C09107=1020.739,297.786,363.988,170.220,49.597,159.600
C09108=1020.733,297.538,364.020,170.215,49.601,159.600
C09109=1020.726,297.291,364.052,170.211,49.603,159.600
C09110=1020.720,297.042,364.084,170.205,49.607,159.600
C09111=1020.713,296.795,364.116,170.200,49.610,159.600
C09112=1020.707,296.547,364.149,170.195,49.613,159.600
C09113=1020.700,296.299,364.180,170.189,49.617,159.600
C09114=1020.694,296.051,364.212,170.184,49.620,159.599
C09115=1020.689,295.804,364.244,170.179,49.623,159.599
C09116=1020.682,295.556,364.276,170.174,49.627,159.599
C09117=1020.676,295.308,364.308,170.168,49.630,159.599
C09118=1020.669,295.061,364.340,170.163,49.633,159.599
C09119=1020.663,294.812,364.372,170.158,49.637,159.599
C09120=1020.657,294.564,364.404,170.153,49.640,159.599
C09121=1020.650,294.316,364.435,170.148,49.643,159.599
C09122=1020.644,294.068,364.467,170.143,49.647,159.599
C09123=1020.638,293.821,364.499,170.138,49.650,159.599
C09124=1020.632,293.592,364.529,170.133,49.653,159.599
C09125=1020.627,293.362,364.558,170.128,49.656,159.599
C09126=1020.620,293.133,364.587,170.123,49.659,159.599
C09127=1020.614,292.904,364.616,170.119,49.662,159.599
C09128=1020.608,292.674,364.645,170.113,49.666,159.599
C09129=1020.603,292.445,364.675,170.110,49.669,159.599
C09130=1020.596,292.216,364.704,170.104,49.673,159.599
C09131=1020.590,291.986,364.732,170.100,49.675,159.599
C09132=1020.584,291.738,364.764,170.095,49.679,159.599
C09133=1020.578,291.490,364.796,170.090,49.683,159.599
C09134=1020.571,291.242,364.827,170.084,49.686,159.599
C09135=1020.565,290.995,364.858,170.079,49.690,159.599
C09136=1020.558,290.747,364.890,170.074,49.693,159.599
C09137=1020.552,290.499,364.921,170.069,49.697,159.599
C09138=1020.545,290.251,364.952,170.064,49.700,159.599
C09139=1020.539,290.004,364.983,170.059,49.704,159.599
C09140=1020.533,289.756,365.015,170.054,49.707,159.599
C09141=1020.526,289.507,365.046,170.049,49.711,159.599
C09142=1020.520,289.259,365.077,170.044,49.715,159.599
C09143=1020.514,289.012,365.108,170.038,49.719,159.599
C09144=1020.507,288.763,365.139,170.034,49.722,159.599
C09145=1020.500,288.515,365.170,170.028,49.726,159.599
C09146=1020.494,288.268,365.202,170.023,49.730,159.599
C09147=1020.488,288.020,365.232,170.018,49.734,159.599
C09148=1020.481,287.772,365.264,170.014,49.736,159.599
C09149=1020.474,287.524,365.295,170.009,49.740,159.599
C09150=1020.469,287.276,365.325,170.004,49.744,159.599
C09151=1020.462,287.028,365.357,169.999,49.748,159.599
C09152=1020.455,286.780,365.388,169.994,49.752,159.599
C09153=1020.449,286.533,365.419,169.989,49.755,159.599
C09154=1020.443,286.284,365.449,169.984,49.759,159.599
C09155=1020.436,286.036,365.481,169.979,49.763,159.599
C09156=1020.430,285.788,365.511,169.974,49.767,159.599
C09157=1020.424,285.540,365.543,169.969,49.771,159.599
C09158=1020.417,285.292,365.573,169.964,49.774,159.599
C09159=1020.411,285.045,365.604,169.959,49.778,159.599
C09160=1020.405,284.796,365.635,169.954,49.782,159.600
C09161=1020.399,284.548,365.665,169.949,49.786,159.599
C09162=1020.392,284.300,365.697,169.944,49.789,159.600
C09163=1020.386,284.052,365.728,169.939,49.793,159.600
C09164=1020.379,283.804,365.757,169.934,49.797,159.600
C09165=1020.373,283.556,365.788,169.929,49.801,159.600
C09166=1020.367,283.309,365.819,169.924,49.805,159.600
C09167=1020.360,283.060,365.850,169.919,49.809,159.600
C09168=1020.354,282.812,365.881,169.914,49.813,159.600
C09169=1020.347,282.564,365.910,169.909,49.817,159.600
C09170=1020.341,282.316,365.942,169.904,49.821,159.600
C09171=1020.335,282.068,365.972,169.899,49.825,159.600
C09172=1020.328,281.820,366.003,169.895,49.829,159.600
C09173=1020.322,281.572,366.033,169.890,49.833,159.600
C09174=1020.315,281.324,366.063,169.886,49.836,159.601
C09175=1020.309,281.076,366.094,169.881,49.840,159.601
C09176=1020.303,280.827,366.124,169.876,49.845,159.601
C09177=1020.297,280.580,366.155,169.871,49.849,159.601
C09178=1020.290,280.332,366.186,169.866,49.853,159.601
C09179=1020.284,280.084,366.216,169.861,49.857,159.601
C09180=1020.278,279.836,366.247,169.856,49.861,159.601
C09181=1020.272,279.588,366.277,169.852,49.865,159.601
C09182=1020.265,279.340,366.307,169.847,49.868,159.602
C09183=1020.259,279.092,366.337,169.842,49.872,159.602
C09184=1020.254,278.869,366.365,169.838,49.876,159.602
C09185=1020.247,278.645,366.392,169.833,49.880,159.602
C09186=1020.242,278.422,366.419,169.829,49.884,159.602
C09187=1020.237,278.199,366.447,169.825,49.887,159.602
C09188=1020.231,277.976,366.474,169.820,49.891,159.602
C09189=1020.226,277.753,366.501,169.816,49.895,159.603
C09190=1020.219,277.529,366.528,169.812,49.898,159.603
C09191=1020.214,277.306,366.556,169.807,49.902,159.603
C09192=1020.209,277.058,366.586,169.802,49.906,159.603
C09193=1020.201,276.810,366.616,169.797,49.910,159.603
C09194=1020.196,276.562,366.647,169.792,49.914,159.603
C09195=1020.189,276.314,366.676,169.788,49.919,159.603
C09196=1020.183,276.066,366.707,169.783,49.923,159.603
C09197=1020.176,275.818,366.736,169.778,49.927,159.604
C09198=1020.171,275.570,366.766,169.774,49.931,159.604
C09199=1020.163,275.322,366.797,169.769,49.935,159.604
C09200=1020.158,275.073,366.826,169.764,49.940,159.604
C09201=1020.152,274.825,366.857,169.759,49.944,159.604
C09202=1020.145,274.577,366.887,169.755,49.948,159.604
C09203=1020.139,274.329,366.916,169.751,49.952,159.605
C09204=1020.133,274.081,366.946,169.746,49.957,159.605
C09205=1020.126,273.833,366.977,169.741,49.961,159.605
C09206=1020.120,273.584,367.006,169.737,49.965,159.605
C09207=1020.114,273.337,367.036,169.732,49.969,159.605
C09208=1020.107,273.088,367.066,169.727,49.974,159.606
C09209=1020.102,272.840,367.096,169.722,49.978,159.606
C09210=1020.095,272.592,367.126,169.718,49.982,159.606
C09211=1020.090,272.344,367.155,169.713,49.986,159.606
C09212=1020.082,272.096,367.185,169.708,49.991,159.606
C09213=1020.076,271.848,367.214,169.704,49.995,159.607
C09214=1020.070,271.600,367.245,169.699,49.999,159.607
C09215=1020.064,271.352,367.274,169.694,50.004,159.607
C09216=1020.058,271.103,367.304,169.690,50.009,159.607
C09217=1020.051,270.855,367.334,169.685,50.013,159.607
C09218=1020.046,270.607,367.363,169.680,50.017,159.608
C09219=1020.039,270.359,367.393,169.676,50.022,159.608
C09220=1020.033,270.111,367.422,169.671,50.026,159.608
C09221=1020.027,269.862,367.453,169.666,50.030,159.608
C09222=1020.020,269.614,367.482,169.662,50.035,159.609
C09223=1020.015,269.366,367.511,169.657,50.039,159.609
C09224=1020.009,269.118,367.540,169.652,50.044,159.609
C09225=1020.002,268.870,367.570,169.648,50.048,159.609
C09226=1019.996,268.622,367.599,169.643,50.053,159.610
C09227=1019.990,268.373,367.629,169.638,50.057,159.610
C09228=1019.984,268.125,367.658,169.634,50.061,159.610
C09229=1019.977,267.877,367.688,169.629,50.066,159.610
C09230=1019.971,267.629,367.718,169.624,50.071,159.610
C09231=1019.965,267.381,367.747,169.620,50.075,159.611
C09232=1019.959,267.133,367.776,169.615,50.080,159.611
C09233=1019.953,266.885,367.805,169.611,50.085,159.611
C09234=1019.946,266.636,367.836,169.606,50.089,159.612
C09235=1019.940,266.388,367.865,169.602,50.094,159.612
C09236=1019.934,266.140,367.894,169.597,50.098,159.612
C09237=1019.928,265.892,367.923,169.593,50.103,159.612
C09238=1019.921,265.643,367.952,169.588,50.107,159.612
C09239=1019.916,265.395,367.981,169.583,50.112,159.613
C09240=1019.910,265.147,368.010,169.579,50.116,159.613
C09241=1019.903,264.899,368.039,169.574,50.121,159.613
C09242=1019.897,264.651,368.068,169.570,50.126,159.614
C09243=1019.891,264.402,368.097,169.565,50.131,159.614
C09244=1019.885,264.182,368.124,169.560,50.135,159.614
C09245=1019.880,263.961,368.149,169.557,50.139,159.615
C09246=1019.874,263.740,368.175,169.553,50.143,159.615
C09247=1019.868,263.519,368.201,169.548,50.147,159.615
C09248=1019.863,263.298,368.227,169.545,50.152,159.615
C09249=1019.857,263.078,368.253,169.541,50.155,159.615
C09250=1019.852,262.856,368.278,169.537,50.160,159.616
C09251=1019.846,262.636,368.304,169.533,50.164,159.616
C09252=1019.841,262.387,368.334,169.528,50.169,159.616
C09253=1019.835,262.139,368.363,169.524,50.174,159.617
C09254=1019.829,261.890,368.391,169.519,50.178,159.617
C09255=1019.822,261.642,368.420,169.515,50.183,159.617
C09256=1019.816,261.394,368.449,169.511,50.188,159.618
C09257=1019.810,261.146,368.478,169.506,50.193,159.618
C09258=1019.804,260.898,368.507,169.502,50.198,159.618
C09259=1019.798,260.649,368.536,169.497,50.202,159.619
C09260=1019.791,260.401,368.565,169.493,50.207,159.619
C09261=1019.785,260.153,368.594,169.488,50.212,159.619
C09262=1019.779,259.905,368.623,169.484,50.217,159.620
C09263=1019.773,259.656,368.651,169.478,50.222,159.620
C09264=1019.766,259.408,368.680,169.474,50.227,159.620
C09265=1019.760,259.159,368.708,169.470,50.232,159.620
C09266=1019.754,258.912,368.737,169.465,50.237,159.621
C09267=1019.748,258.664,368.764,169.461,50.242,159.621
C09268=1019.741,258.415,368.793,169.457,50.247,159.622
C09269=1019.736,258.167,368.822,169.452,50.252,159.622
C09270=1019.729,257.919,368.850,169.448,50.257,159.622
C09271=1019.723,257.670,368.879,169.444,50.262,159.623
C09272=1019.716,257.422,368.908,169.438,50.267,159.623
C09273=1019.710,257.173,368.935,169.434,50.272,159.623
C09274=1019.703,256.925,368.964,169.430,50.277,159.624
C09275=1019.697,256.677,368.993,169.425,50.282,159.624
C09276=1019.690,256.429,369.021,169.421,50.287,159.625
C09277=1019.685,256.180,369.049,169.417,50.293,159.625
C09278=1019.679,255.932,369.077,169.412,50.297,159.625
C09279=1019.672,255.684,369.106,169.408,50.303,159.626
C09280=1019.666,255.435,369.134,169.403,50.308,159.626
C09281=1019.660,255.187,369.162,169.399,50.313,159.627
C09282=1019.653,254.939,369.191,169.394,50.318,159.627
C09283=1019.647,254.690,369.219,169.390,50.323,159.627
C09284=1019.642,254.442,369.247,169.386,50.328,159.628
C09285=1019.635,254.194,369.276,169.381,50.333,159.628
C09286=1019.629,253.945,369.304,169.377,50.338,159.628
C09287=1019.623,253.697,369.332,169.373,50.343,159.629
C09288=1019.616,253.448,369.360,169.368,50.348,159.629
C09289=1019.611,253.201,369.389,169.363,50.354,159.630
C09290=1019.605,252.952,369.417,169.359,50.359,159.630
C09291=1019.598,252.704,369.445,169.355,50.364,159.631
C09292=1019.592,252.455,369.473,169.350,50.369,159.631
C09293=1019.586,252.207,369.502,169.346,50.374,159.631
C09294=1019.580,251.959,369.530,169.342,50.380,159.632
C09295=1019.574,251.710,369.558,169.338,50.385,159.632
C09296=1019.568,251.461,369.586,169.333,50.390,159.633
C09297=1019.562,251.214,369.614,169.329,50.395,159.633
C09298=1019.556,250.966,369.643,169.324,50.401,159.633
C09299=1019.550,250.717,369.671,169.320,50.406,159.634
C09300=1019.543,250.468,369.699,169.316,50.411,159.634
C09301=1019.538,250.220,369.727,169.311,50.416,159.635
C09302=1019.532,249.972,369.755,169.307,50.422,159.635
C09303=1019.525,249.723,369.783,169.303,50.427,159.636
C09304=1019.520,249.502,369.808,169.299,50.432,159.636
C09305=1019.515,249.280,369.833,169.295,50.437,159.636
C09306=1019.510,249.058,369.857,169.292,50.441,159.637
C09307=1019.504,248.837,369.883,169.287,50.446,159.637
C09308=1019.499,248.614,369.908,169.284,50.451,159.638
C09309=1019.493,248.393,369.933,169.280,50.455,159.638
C09310=1019.488,248.171,369.958,169.276,50.460,159.638
C09311=1019.483,247.950,369.983,169.272,50.465,159.639
C09312=1019.476,247.702,370.011,169.268,50.470,159.639
C09313=1019.471,247.454,370.039,169.264,50.476,159.640
C09314=1019.464,247.205,370.067,169.260,50.481,159.640
C09315=1019.458,246.956,370.094,169.256,50.486,159.641
C09316=1019.453,246.708,370.122,169.251,50.491,159.641
C09317=1019.446,246.459,370.150,169.247,50.496,159.641
C09318=1019.441,246.211,370.178,169.242,50.502,159.642
C09319=1019.435,245.962,370.206,169.238,50.508,159.642
C09320=1019.429,245.714,370.234,169.234,50.513,159.643
C09321=1019.423,245.466,370.262,169.229,50.518,159.643
C09322=1019.417,245.217,370.290,169.225,50.524,159.643
C09323=1019.411,244.969,370.318,169.221,50.529,159.644
C09324=1019.405,244.721,370.346,169.217,50.534,159.644
C09325=1019.399,244.473,370.373,169.213,50.540,159.645
C09326=1019.393,244.224,370.401,169.209,50.546,159.646
C09327=1019.388,243.976,370.429,169.204,50.551,159.646
C09328=1019.381,243.727,370.457,169.200,50.557,159.646
C09329=1019.376,243.479,370.485,169.196,50.562,159.647
C09330=1019.370,243.230,370.513,169.192,50.567,159.647
C09331=1019.364,242.982,370.540,169.188,50.573,159.648
C09332=1019.358,242.733,370.567,169.184,50.578,159.648
C09333=1019.352,242.485,370.595,169.180,50.584,159.649
C09334=1019.346,242.236,370.622,169.175,50.590,159.649
C09335=1019.340,241.989,370.650,169.171,50.595,159.650
C09336=1019.334,241.740,370.678,169.166,50.601,159.650
C09337=1019.328,241.492,370.705,169.163,50.607,159.651
C09338=1019.322,241.243,370.732,169.159,50.612,159.651
C09339=1019.316,240.994,370.760,169.153,50.618,159.652
C09340=1019.310,240.746,370.787,169.150,50.624,159.652
C09341=1019.304,240.498,370.815,169.146,50.629,159.653
C09342=1019.298,240.249,370.842,169.141,50.635,159.653
C09343=1019.292,240.001,370.870,169.138,50.641,159.654
C09344=1019.286,239.753,370.896,169.133,50.646,159.654
C09345=1019.280,239.504,370.925,169.129,50.652,159.655
C09346=1019.275,239.256,370.951,169.125,50.658,159.656
C09347=1019.268,239.007,370.979,169.121,50.663,159.656
C09348=1019.262,238.759,371.006,169.117,50.669,159.657
C09349=1019.256,238.510,371.034,169.112,50.675,159.657
C09350=1019.250,238.262,371.061,169.108,50.681,159.658
C09351=1019.245,238.013,371.087,169.104,50.686,159.658
C09352=1019.238,237.765,371.115,169.100,50.692,159.659
C09353=1019.232,237.517,371.142,169.095,50.698,159.659
C09354=1019.226,237.268,371.169,169.091,50.704,159.660
C09355=1019.220,237.020,371.196,169.087,50.710,159.660
C09356=1019.214,236.771,371.223,169.083,50.716,159.661
C09357=1019.208,236.522,371.250,169.079,50.722,159.662
C09358=1019.202,236.274,371.276,169.075,50.727,159.662
C09359=1019.195,236.026,371.304,169.071,50.734,159.663
C09360=1019.189,235.777,371.331,169.066,50.739,159.663
C09361=1019.184,235.529,371.357,169.062,50.745,159.664
C09362=1019.177,235.280,371.384,169.059,50.751,159.664
C09363=1019.171,235.032,371.412,169.054,50.757,159.665
C09364=1019.166,234.807,371.436,169.051,50.763,159.666
C09365=1019.160,234.581,371.460,169.047,50.768,159.666
C09366=1019.155,234.356,371.485,169.043,50.774,159.667
C09367=1019.150,234.132,371.509,169.039,50.779,159.667
C09368=1019.145,233.907,371.533,169.035,50.784,159.668
C09369=1019.139,233.682,371.558,169.031,50.790,159.668
C09370=1019.134,233.457,371.582,169.029,50.795,159.669
C09371=1019.128,233.232,371.606,169.024,50.801,159.669
C09372=1019.122,232.983,371.633,169.021,50.807,159.670
C09373=1019.116,232.735,371.660,169.016,50.812,159.670
C09374=1019.110,232.487,371.686,169.012,50.819,159.671
C09375=1019.104,232.238,371.713,169.008,50.825,159.672
C09376=1019.098,231.989,371.740,169.004,50.831,159.672
C09377=1019.092,231.741,371.767,169.000,50.837,159.673
C09378=1019.086,231.493,371.794,168.996,50.843,159.673
C09379=1019.080,231.245,371.821,168.992,50.849,159.674
C09380=1019.074,230.996,371.848,168.987,50.855,159.675
C09381=1019.068,230.747,371.874,168.984,50.861,159.675
C09382=1019.062,230.499,371.901,168.980,50.867,159.676
C09383=1019.057,230.251,371.928,168.975,50.874,159.676
C09384=1019.050,230.001,371.955,168.972,50.880,159.677
C09385=1019.044,229.753,371.981,168.968,50.886,159.678
C09386=1019.039,229.504,372.007,168.963,50.892,159.678
C09387=1019.033,229.256,372.034,168.959,50.898,159.679
C09388=1019.027,229.007,372.061,168.955,50.904,159.680
C09389=1019.020,228.759,372.087,168.951,50.910,159.680
C09390=1019.015,228.510,372.114,168.947,50.916,159.681
C09391=1019.009,228.262,372.140,168.943,50.922,159.681
C09392=1019.003,228.014,372.167,168.939,50.929,159.682
C09393=1018.997,227.765,372.194,168.935,50.935,159.683
C09394=1018.992,227.516,372.220,168.932,50.942,159.684
C09395=1018.985,227.268,372.246,168.927,50.948,159.684
C09396=1018.979,227.019,372.273,168.923,50.954,159.685
C09397=1018.973,226.771,372.299,168.919,50.961,159.685
C09398=1018.968,226.522,372.325,168.915,50.967,159.686
C09399=1018.961,226.274,372.351,168.911,50.973,159.687
C09400=1018.955,226.025,372.378,168.906,50.979,159.687
C09401=1018.950,225.777,372.405,168.903,50.985,159.688
C09402=1018.943,225.528,372.430,168.899,50.993,159.689
C09403=1018.937,225.279,372.457,168.895,50.999,159.689
C09404=1018.931,225.031,372.482,168.890,51.005,159.690
C09405=1018.925,224.782,372.509,168.886,51.011,159.691
C09406=1018.919,224.534,372.536,168.883,51.018,159.692
C09407=1018.913,224.285,372.561,168.879,51.024,159.692
C09408=1018.907,224.037,372.588,168.875,51.031,159.693
C09409=1018.901,223.788,372.613,168.871,51.038,159.694
C09410=1018.895,223.539,372.640,168.867,51.044,159.694
C09411=1018.889,223.290,372.666,168.862,51.050,159.695
C09412=1018.883,223.042,372.692,168.859,51.056,159.695
C09413=1018.877,222.793,372.718,168.855,51.063,159.696
C09414=1018.871,222.545,372.744,168.851,51.070,159.697
C09415=1018.865,222.296,372.770,168.847,51.076,159.698
C09416=1018.859,222.048,372.796,168.843,51.083,159.698
C09417=1018.853,221.799,372.822,168.839,51.089,159.699
C09418=1018.847,221.551,372.848,168.835,51.096,159.700
C09419=1018.841,221.302,372.874,168.831,51.102,159.700
C09420=1018.835,221.054,372.900,168.826,51.109,159.701
C09421=1018.830,220.805,372.926,168.823,51.116,159.702
C09422=1018.824,220.557,372.952,168.818,51.122,159.702
C09423=1018.818,220.308,372.978,168.815,51.129,159.703
C09424=1018.812,220.079,373.002,168.811,51.135,159.704
C09425=1018.807,219.850,373.026,168.808,51.141,159.705
C09426=1018.801,219.621,373.050,168.804,51.147,159.705
C09427=1018.796,219.392,373.074,168.801,51.153,159.706
C09428=1018.790,219.163,373.098,168.796,51.159,159.706
C09429=1018.785,218.933,373.122,168.793,51.165,159.707
C09430=1018.779,218.704,373.146,168.789,51.171,159.708
C09431=1018.774,218.475,373.170,168.785,51.177,159.708
C09432=1018.768,218.226,373.196,168.782,51.184,159.709
C09433=1018.762,217.978,373.221,168.778,51.191,159.710
C09434=1018.757,217.730,373.246,168.774,51.197,159.711
C09435=1018.750,217.482,373.272,168.770,51.204,159.712
C09436=1018.745,217.233,373.298,168.767,51.211,159.712
C09437=1018.738,216.984,373.324,168.762,51.218,159.713
C09438=1018.732,216.735,373.349,168.758,51.225,159.714
C09439=1018.727,216.486,373.375,168.755,51.232,159.715
C09440=1018.720,216.238,373.401,168.750,51.238,159.715
C09441=1018.714,215.990,373.426,168.747,51.245,159.716
C09442=1018.708,215.741,373.452,168.742,51.252,159.717
C09443=1018.702,215.492,373.478,168.739,51.259,159.718
C09444=1018.696,215.243,373.503,168.735,51.265,159.718
C09445=1018.690,214.995,373.528,168.730,51.273,159.719
C09446=1018.684,214.746,373.554,168.727,51.279,159.720
C09447=1018.678,214.497,373.580,168.723,51.287,159.721
C09448=1018.673,214.249,373.605,168.720,51.293,159.722
C09449=1018.666,214.000,373.630,168.715,51.300,159.722
C09450=1018.661,213.752,373.657,168.712,51.307,159.723
C09451=1018.654,213.503,373.682,168.707,51.314,159.724
C09452=1018.648,213.255,373.707,168.703,51.321,159.725
C09453=1018.643,213.006,373.733,168.700,51.328,159.725
C09454=1018.637,212.757,373.759,168.696,51.335,159.726
C09455=1018.630,212.508,373.784,168.692,51.341,159.727
C09456=1018.625,212.260,373.809,168.688,51.349,159.728
C09457=1018.619,212.011,373.835,168.684,51.356,159.728
C09458=1018.613,211.763,373.860,168.680,51.363,159.729
C09459=1018.607,211.514,373.885,168.676,51.370,159.730
C09460=1018.601,211.265,373.911,168.673,51.377,159.731
C09461=1018.596,211.017,373.936,168.669,51.384,159.732
C09462=1018.590,210.768,373.962,168.664,51.391,159.733
C09463=1018.584,210.519,373.986,168.661,51.398,159.733
C09464=1018.578,210.270,374.012,168.657,51.405,159.734
C09465=1018.572,210.021,374.038,168.654,51.412,159.735
C09466=1018.566,209.774,374.063,168.650,51.419,159.736
C09467=1018.560,209.525,374.088,168.645,51.426,159.737
C09468=1018.554,209.276,374.113,168.642,51.433,159.738
C09469=1018.548,209.028,374.139,168.638,51.440,159.738
C09470=1018.542,208.778,374.163,168.634,51.448,159.739
C09471=1018.537,208.530,374.189,168.631,51.454,159.740
C09472=1018.531,208.281,374.214,168.626,51.462,159.741
C09473=1018.525,208.033,374.239,168.622,51.469,159.741
C09474=1018.518,207.784,374.265,168.618,51.477,159.742
C09475=1018.513,207.535,374.289,168.615,51.484,159.743
C09476=1018.507,207.287,374.314,168.611,51.491,159.744
C09477=1018.501,207.038,374.340,168.607,51.498,159.745
C09478=1018.495,206.789,374.364,168.603,51.505,159.746
C09479=1018.489,206.541,374.389,168.600,51.513,159.747
C09480=1018.483,206.292,374.415,168.595,51.520,159.748
C09481=1018.477,206.043,374.439,168.591,51.527,159.748
C09482=1018.472,205.795,374.464,168.588,51.534,159.749
C09483=1018.465,205.546,374.490,168.584,51.542,159.750
C09484=1018.460,205.317,374.512,168.581,51.548,159.751
C09485=1018.454,205.087,374.535,168.577,51.555,159.752
C09486=1018.449,204.858,374.559,168.573,51.562,159.752
C09487=1018.444,204.629,374.581,168.570,51.569,159.753
C09488=1018.438,204.400,374.603,168.566,51.575,159.754
C09489=1018.432,204.171,374.626,168.563,51.582,159.755
C09490=1018.426,203.942,374.650,168.559,51.589,159.756
C09491=1018.400,202.697,374.768,168.087,51.498,159.649
C09492=1018.396,202.448,374.791,168.082,51.506,159.650
C09493=1018.390,202.199,374.814,168.078,51.514,159.651
C09494=1018.385,201.950,374.837,168.073,51.523,159.652
C09495=1018.381,201.701,374.860,168.069,51.532,159.653
C09496=1018.376,201.452,374.883,168.064,51.540,159.653
C09497=1018.371,201.204,374.906,168.060,51.548,159.654
C09498=1018.366,200.954,374.929,168.055,51.556,159.655
C09499=1018.361,200.705,374.953,168.051,51.565,159.656
C09500=1018.356,200.457,374.976,168.046,51.573,159.657
C09501=1018.351,200.208,374.999,168.041,51.582,159.658
C09502=1018.346,199.959,375.022,168.037,51.590,159.659
C09503=1018.341,199.710,375.045,168.033,51.599,159.660
C09504=1018.336,199.461,375.069,168.028,51.607,159.661
C09505=1018.332,199.212,375.091,168.023,51.616,159.662
C09506=1018.326,198.963,375.114,168.019,51.624,159.663
C09507=1018.321,198.715,375.137,168.014,51.632,159.663
C09508=1018.316,198.465,375.160,168.010,51.641,159.664
C09509=1018.311,198.217,375.182,168.005,51.649,159.665
C09510=1018.305,197.968,375.205,168.001,51.658,159.666
C09511=1018.301,197.718,375.228,167.997,51.666,159.667
C09512=1018.295,197.470,375.250,167.992,51.675,159.668
C09513=1018.290,197.221,375.273,167.988,51.684,159.669
C09514=1018.286,196.972,375.296,167.983,51.693,159.670
C09515=1018.280,196.723,375.319,167.978,51.701,159.671
C09516=1018.275,196.474,375.341,167.975,51.710,159.672
C09517=1018.270,196.225,375.364,167.970,51.718,159.673
C09518=1018.265,195.976,375.386,167.966,51.727,159.674
C09519=1018.259,195.727,375.409,167.961,51.735,159.675
C09520=1018.254,195.479,375.432,167.956,51.744,159.676
C09521=1018.250,195.229,375.454,167.953,51.752,159.677
C09522=1018.245,194.981,375.477,167.948,51.761,159.678
C09523=1018.239,194.732,375.499,167.943,51.770,159.678
C09524=1018.235,194.483,375.522,167.939,51.779,159.679
C09525=1018.229,194.234,375.545,167.935,51.787,159.680
C09526=1018.224,193.985,375.567,167.931,51.796,159.681
C09527=1018.219,193.736,375.590,167.926,51.804,159.682
C09528=1018.215,193.487,375.612,167.922,51.813,159.683
C09529=1018.210,193.239,375.635,167.918,51.821,159.684
C09530=1018.205,192.989,375.657,167.913,51.830,159.685
C09531=1018.200,192.741,375.680,167.908,51.838,159.686
C09532=1018.194,192.491,375.702,167.905,51.847,159.687
C09533=1018.189,192.243,375.725,167.900,51.856,159.688
C09534=1018.185,191.994,375.747,167.896,51.865,159.689
C09535=1018.180,191.744,375.769,167.892,51.873,159.690
C09536=1018.175,191.496,375.792,167.887,51.882,159.691
C09537=1018.170,191.246,375.815,167.883,51.890,159.692
C09538=1018.165,190.998,375.837,167.879,51.899,159.693
C09539=1018.160,190.749,375.859,167.874,51.907,159.694
C09540=1018.155,190.499,375.882,167.870,51.916,159.695
C09541=1018.150,190.251,375.905,167.866,51.924,159.696
C09542=1018.145,190.002,375.927,167.862,51.933,159.697
C09543=1018.140,189.753,375.949,167.857,51.941,159.698
C09544=1018.136,189.504,375.971,167.854,51.950,159.699
C09545=1018.131,189.256,375.994,167.849,51.959,159.699
C09546=1018.125,189.006,376.016,167.845,51.968,159.701
C09547=1018.121,188.757,376.038,167.841,51.976,159.702
C09548=1018.116,188.509,376.061,167.836,51.985,159.702
C09549=1018.111,188.259,376.083,167.832,51.994,159.704
C09550=1018.106,188.010,376.106,167.828,52.002,159.704
C09551=1018.102,187.761,376.128,167.824,52.011,159.705
C09552=1018.096,187.481,376.153,167.819,52.020,159.706
C09553=1018.090,187.199,376.178,167.814,52.030,159.708
C09554=1018.085,186.919,376.203,167.810,52.039,159.709
C09555=1018.080,186.638,376.228,167.805,52.049,159.710
C09556=1018.075,186.390,376.251,167.801,52.058,159.711
C09557=1018.070,186.140,376.273,167.797,52.066,159.712
C09558=1018.065,185.892,376.295,167.793,52.075,159.713
C09559=1018.060,185.643,376.317,167.789,52.083,159.714
C09560=1018.055,185.394,376.339,167.785,52.093,159.715
C09561=1018.051,185.145,376.361,167.781,52.101,159.716
C09562=1018.046,184.896,376.384,167.776,52.110,159.717
C09563=1018.041,184.647,376.406,167.772,52.118,159.717
C09564=1018.037,184.398,376.429,167.768,52.127,159.719
C09565=1018.032,184.149,376.451,167.764,52.135,159.719
C09566=1018.027,183.900,376.472,167.760,52.144,159.721
C09567=1018.022,183.651,376.495,167.755,52.152,159.721
C09568=1018.018,183.402,376.517,167.752,52.161,159.723
C09569=1018.013,183.153,376.539,167.747,52.170,159.723
C09570=1018.008,182.904,376.561,167.744,52.178,159.724
C09571=1018.003,182.655,376.583,167.739,52.187,159.725
C09572=1017.999,182.406,376.605,167.736,52.195,159.726
C09573=1017.994,182.157,376.627,167.731,52.204,159.727
C09574=1017.989,181.908,376.649,167.728,52.213,159.728
C09575=1017.984,181.659,376.671,167.723,52.222,159.729
C09576=1017.979,181.410,376.693,167.719,52.231,159.730
C09577=1017.974,181.161,376.714,167.715,52.239,159.731
C09578=1017.968,180.912,376.736,167.711,52.248,159.732
C09579=1017.964,180.663,376.758,167.707,52.257,159.733
C09580=1017.958,180.414,376.778,167.703,52.266,159.735
C09581=1017.954,180.165,376.800,167.699,52.275,159.736
C09582=1017.949,179.916,376.822,167.695,52.284,159.737
C09583=1017.943,179.667,376.842,167.692,52.293,159.738
C09584=1017.938,179.417,376.865,167.687,52.301,159.739
C09585=1017.934,179.168,376.886,167.682,52.310,159.740
C09586=1017.928,178.919,376.907,167.679,52.319,159.741
C09587=1017.923,178.671,376.929,167.675,52.328,159.742
C09588=1017.918,178.422,376.949,167.672,52.337,159.743
C09589=1017.913,178.173,376.971,167.667,52.346,159.744
C09590=1017.909,177.923,376.993,167.663,52.355,159.745
C09591=1017.903,177.675,377.014,167.659,52.364,159.746
C09592=1017.898,177.426,377.036,167.655,52.373,159.747
C09593=1017.893,177.176,377.057,167.651,52.382,159.748
C09594=1017.887,176.927,377.078,167.647,52.391,159.749
C09595=1017.883,176.678,377.100,167.643,52.400,159.750
C09596=1017.878,176.429,377.121,167.640,52.409,159.751
C09597=1017.873,176.180,377.142,167.635,52.418,159.752
C09598=1017.868,175.931,377.164,167.631,52.426,159.753
C09599=1017.863,175.682,377.184,167.627,52.435,159.754
C09600=1017.858,175.433,377.206,167.623,52.444,159.755
C09601=1017.853,175.184,377.227,167.620,52.453,159.756
C09602=1017.848,174.935,377.249,167.616,52.462,159.757
C09603=1017.843,174.686,377.270,167.612,52.471,159.759
C09604=1017.839,174.437,377.292,167.608,52.480,159.760
C09605=1017.833,174.188,377.312,167.603,52.488,159.760
C09606=1017.828,173.939,377.334,167.600,52.497,159.762
C09607=1017.823,173.690,377.355,167.596,52.506,159.763
C09608=1017.819,173.440,377.376,167.593,52.515,159.764
C09609=1017.814,173.192,377.398,167.588,52.524,159.765
C09610=1017.809,172.943,377.418,167.585,52.533,159.766
C09611=1017.804,172.694,377.440,167.580,52.542,159.767
C09612=1017.799,172.445,377.461,167.577,52.551,159.768
C09613=1017.794,172.195,377.482,167.573,52.560,159.769
C09614=1017.789,171.946,377.504,167.570,52.569,159.770
C09615=1017.784,171.697,377.524,167.565,52.578,159.771
C09616=1017.779,171.416,377.548,167.562,52.588,159.772
C09617=1017.773,171.135,377.572,167.557,52.598,159.773
C09618=1017.768,170.854,377.596,167.553,52.608,159.775
C09619=1017.762,170.573,377.620,167.548,52.618,159.776
C09620=1017.757,170.324,377.641,167.545,52.627,159.777
C09621=1017.753,170.075,377.662,167.540,52.635,159.778
C09622=1017.748,169.826,377.684,167.537,52.644,159.779
C09623=1017.743,169.577,377.704,167.533,52.653,159.780
C09624=1017.738,169.327,377.725,167.529,52.662,159.781
C09625=1017.733,169.079,377.746,167.525,52.671,159.782
C09626=1017.729,168.830,377.767,167.522,52.680,159.783
C09627=1017.724,168.581,377.789,167.517,52.689,159.784
C09628=1017.719,168.332,377.809,167.514,52.698,159.785
C09629=1017.714,168.082,377.830,167.511,52.706,159.786
C09630=1017.709,167.833,377.852,167.507,52.716,159.787
C09631=1017.704,167.584,377.873,167.503,52.724,159.789
C09632=1017.700,167.335,377.893,167.499,52.734,159.790
C09633=1017.695,167.086,377.914,167.495,52.742,159.791
C09634=1017.690,166.838,377.936,167.491,52.751,159.792
C09635=1017.686,166.588,377.957,167.488,52.760,159.793
C09636=1017.680,166.339,377.978,167.485,52.769,159.794
C09637=1017.676,166.090,377.999,167.481,52.778,159.795
C09638=1017.671,165.841,378.019,167.477,52.787,159.796
C09639=1017.667,165.592,378.040,167.473,52.795,159.797
C09640=1017.662,165.343,378.062,167.470,52.804,159.798
C09641=1017.657,165.094,378.083,167.466,52.813,159.799
C09642=1017.652,164.844,378.104,167.462,52.822,159.800
C09643=1017.648,164.596,378.124,167.459,52.831,159.801
C09644=1017.643,164.346,378.145,167.454,52.840,159.802
C09645=1017.638,164.097,378.166,167.451,52.849,159.803
C09646=1017.633,163.848,378.187,167.448,52.857,159.804
C09647=1017.629,163.599,378.207,167.444,52.867,159.806
C09648=1017.624,163.351,378.229,167.441,52.876,159.807
C09649=1017.619,163.101,378.250,167.437,52.884,159.808
C09650=1017.615,162.852,378.271,167.433,52.893,159.809
C09651=1017.610,162.603,378.291,167.430,52.902,159.810
C09652=1017.606,162.354,378.312,167.426,52.911,159.811
C09653=1017.600,162.105,378.333,167.422,52.920,159.812
C09654=1017.596,161.855,378.354,167.419,52.928,159.813
C09655=1017.591,161.607,378.374,167.415,52.937,159.814
C09656=1017.587,161.358,378.395,167.411,52.946,159.815
C09657=1017.582,161.108,378.417,167.408,52.955,159.816
C09658=1017.577,160.860,378.437,167.405,52.964,159.817
C09659=1017.573,160.610,378.458,167.400,52.973,159.818
C09660=1017.568,160.361,378.478,167.397,52.982,159.819
C09661=1017.563,160.112,378.500,167.394,52.990,159.820
C09662=1017.559,159.863,378.520,167.390,53.000,159.822
C09663=1017.554,159.614,378.541,167.386,53.008,159.822
C09664=1017.549,159.364,378.562,167.383,53.017,159.824
C09665=1017.545,159.116,378.582,167.380,53.026,159.825
C09666=1017.540,158.867,378.603,167.376,53.035,159.826
C09667=1017.536,158.617,378.625,167.373,53.044,159.827
C09668=1017.531,158.368,378.644,167.369,53.053,159.828
C09669=1017.526,158.119,378.665,167.365,53.062,159.829
C09670=1017.521,157.870,378.685,167.362,53.071,159.830
C09671=1017.516,157.621,378.705,167.358,53.080,159.831
C09672=1017.511,157.372,378.725,167.355,53.089,159.832
C09673=1017.506,157.123,378.746,167.352,53.098,159.834
C09674=1017.501,156.874,378.766,167.348,53.107,159.835
C09675=1017.497,156.624,378.786,167.344,53.116,159.836
C09676=1017.492,156.375,378.807,167.340,53.126,159.837
C09677=1017.487,156.126,378.827,167.337,53.135,159.838
C09678=1017.482,155.877,378.847,167.334,53.143,159.839
C09679=1017.477,155.628,378.867,167.330,53.153,159.840
C09680=1017.472,155.347,378.889,167.326,53.163,159.841
C09681=1017.467,155.065,378.913,167.322,53.173,159.843
C09682=1017.461,154.784,378.935,167.318,53.183,159.844
C09683=1017.456,154.503,378.959,167.314,53.193,159.845
C09684=1017.452,154.254,378.978,167.310,53.202,159.846
C09685=1017.446,154.004,378.999,167.307,53.211,159.847
C09686=1017.441,153.755,379.020,167.304,53.220,159.848
C09687=1017.437,153.506,379.039,167.300,53.230,159.850
C09688=1017.431,153.257,379.060,167.297,53.239,159.851
C09689=1017.427,153.008,379.079,167.293,53.247,159.852
C09690=1017.422,152.759,379.100,167.289,53.257,159.853
C09691=1017.417,152.509,379.119,167.286,53.266,159.854
C09692=1017.412,152.261,379.140,167.283,53.275,159.855
C09693=1017.407,152.011,379.159,167.279,53.284,159.856
C09694=1017.403,151.763,379.180,167.276,53.294,159.858
C09695=1017.398,151.513,379.199,167.272,53.303,159.859
C09696=1017.393,151.264,379.219,167.269,53.312,159.860
C09697=1017.388,151.015,379.240,167.266,53.321,159.861
C09698=1017.383,150.765,379.259,167.262,53.330,159.862
C09699=1017.378,150.517,379.280,167.259,53.339,159.863
C09700=1017.373,150.267,379.299,167.256,53.348,159.864
C09701=1017.369,150.018,379.319,167.252,53.357,159.865
C09702=1017.364,149.769,379.339,167.249,53.366,159.867
C09703=1017.360,149.520,379.359,167.246,53.375,159.868
C09704=1017.354,149.270,379.379,167.242,53.385,159.869
C09705=1017.350,149.021,379.399,167.238,53.394,159.870
C09706=1017.345,148.772,379.419,167.235,53.403,159.871
C09707=1017.340,148.523,379.439,167.231,53.412,159.872
C09708=1017.335,148.273,379.459,167.228,53.421,159.873
C09709=1017.330,148.025,379.478,167.225,53.430,159.874
C09710=1017.325,147.776,379.498,167.221,53.439,159.875
C09711=1017.321,147.527,379.518,167.218,53.448,159.877
C09712=1017.316,147.277,379.538,167.215,53.457,159.878
C09713=1017.311,147.028,379.557,167.211,53.467,159.879
C09714=1017.306,146.779,379.578,167.208,53.476,159.880
C09715=1017.302,146.530,379.597,167.205,53.485,159.881
C09716=1017.297,146.280,379.617,167.201,53.495,159.882
C09717=1017.292,146.031,379.636,167.198,53.504,159.884
C09718=1017.286,145.782,379.656,167.195,53.513,159.885
C09719=1017.282,145.533,379.676,167.191,53.522,159.886
C09720=1017.278,145.284,379.695,167.188,53.531,159.887
C09721=1017.273,145.034,379.715,167.185,53.540,159.888
C09722=1017.268,144.785,379.734,167.181,53.549,159.889
C09723=1017.263,144.536,379.754,167.178,53.558,159.890
C09724=1017.258,144.287,379.774,167.175,53.567,159.892
C09725=1017.252,144.038,379.793,167.171,53.577,159.893
C09726=1017.248,143.789,379.813,167.168,53.586,159.894
C09727=1017.243,143.539,379.833,167.165,53.595,159.895
C09728=1017.238,143.290,379.851,167.161,53.605,159.896
C09729=1017.234,143.041,379.871,167.158,53.614,159.897
C09730=1017.229,142.792,379.891,167.155,53.623,159.898
C09731=1017.224,142.543,379.910,167.151,53.632,159.900
C09732=1017.219,142.293,379.929,167.148,53.641,159.901
C09733=1017.214,142.044,379.949,167.145,53.651,159.902
C09734=1017.210,141.795,379.968,167.141,53.660,159.903
C09735=1017.204,141.546,379.988,167.138,53.669,159.904
C09736=1017.200,141.297,380.007,167.135,53.678,159.905
C09737=1017.195,141.047,380.027,167.131,53.688,159.907
C09738=1017.190,140.798,380.046,167.128,53.697,159.908
C09739=1017.186,140.549,380.065,167.125,53.706,159.909
C09740=1017.181,140.299,380.085,167.122,53.715,159.910
C09741=1017.176,140.051,380.104,167.118,53.724,159.911
C09742=1017.171,139.802,380.123,167.115,53.733,159.912
C09743=1017.166,139.552,380.143,167.113,53.743,159.914
C09744=1017.161,139.271,380.165,167.108,53.753,159.915
C09745=1017.155,138.990,380.187,167.105,53.763,159.916
C09746=1017.150,138.708,380.208,167.101,53.774,159.917
C09747=1017.144,138.426,380.230,167.098,53.784,159.919
C09748=1017.140,138.177,380.250,167.095,53.793,159.920
C09749=1017.135,137.929,380.269,167.091,53.803,159.921
C09750=1017.130,137.679,380.289,167.088,53.812,159.922
C09751=1017.125,137.430,380.308,167.085,53.821,159.923
C09752=1017.121,137.181,380.326,167.081,53.830,159.924
C09753=1017.115,136.931,380.346,167.078,53.839,159.926
C09754=1017.111,136.682,380.365,167.075,53.848,159.927
C09755=1017.106,136.433,380.384,167.073,53.858,159.928
C09756=1017.101,136.184,380.404,167.069,53.868,159.929
C09757=1017.096,135.934,380.422,167.066,53.877,159.930
C09758=1017.092,135.685,380.441,167.063,53.886,159.932
C09759=1017.087,135.436,380.460,167.059,53.895,159.933
C09760=1017.082,135.187,380.480,167.056,53.904,159.934
C09761=1017.077,134.937,380.498,167.053,53.914,159.935
C09762=1017.073,134.688,380.518,167.049,53.923,159.936
C09763=1017.067,134.439,380.537,167.046,53.932,159.937
C09764=1017.062,134.190,380.556,167.043,53.941,159.939
C09765=1017.058,133.941,380.575,167.041,53.951,159.940
C09766=1017.053,133.692,380.593,167.037,53.960,159.941
C09767=1017.048,133.442,380.613,167.034,53.970,159.942
C09768=1017.043,133.193,380.631,167.031,53.979,159.943
C09769=1017.038,132.944,380.650,167.027,53.988,159.945
C09770=1017.033,132.695,380.670,167.024,53.997,159.946
C09771=1017.028,132.445,380.688,167.021,54.006,159.947
C09772=1017.024,132.196,380.708,167.018,54.015,159.948
C09773=1017.019,131.947,380.727,167.014,54.025,159.949
C09774=1017.014,131.698,380.745,167.012,54.035,159.951
C09775=1017.010,131.449,380.764,167.009,54.044,159.952
C09776=1017.004,131.199,380.783,167.006,54.053,159.953
C09777=1017.000,130.950,380.802,167.002,54.062,159.954
C09778=1016.995,130.701,380.821,166.999,54.071,159.955
C09779=1016.990,130.452,380.839,166.996,54.080,159.956
C09780=1016.985,130.202,380.859,166.993,54.090,159.957
C09781=1016.980,129.952,380.877,166.989,54.099,159.959
C09782=1016.976,129.703,380.897,166.987,54.109,159.960
C09783=1016.971,129.454,380.915,166.984,54.118,159.961
C09784=1016.965,129.205,380.934,166.981,54.127,159.962
C09785=1016.961,128.955,380.952,166.977,54.136,159.963
C09786=1016.956,128.707,380.971,166.975,54.146,159.965
C09787=1016.951,128.457,380.989,166.972,54.155,159.966
C09788=1016.946,128.208,381.008,166.968,54.165,159.967
C09789=1016.941,127.959,381.026,166.966,54.175,159.968
C09790=1016.936,127.709,381.045,166.963,54.184,159.970
C09791=1016.931,127.460,381.063,166.959,54.193,159.971
C09792=1016.926,127.211,381.082,166.956,54.202,159.972
C09793=1016.921,126.962,381.100,166.953,54.212,159.973
C09794=1016.917,126.712,381.119,166.950,54.222,159.974
C09795=1016.912,126.463,381.138,166.947,54.231,159.976
C09796=1016.906,126.213,381.156,166.944,54.240,159.977
C09797=1016.902,125.964,381.175,166.940,54.250,159.978
C09798=1016.896,125.715,381.193,166.937,54.259,159.979
C09799=1016.892,125.466,381.212,166.935,54.268,159.980
C09800=1016.887,125.216,381.230,166.931,54.278,159.982
C09801=1016.882,124.968,381.249,166.928,54.288,159.983
C09802=1016.877,124.718,381.267,166.925,54.297,159.984
C09803=1016.872,124.469,381.285,166.923,54.306,159.985
C09804=1016.867,124.219,381.303,166.919,54.315,159.986
C09805=1016.862,123.970,381.322,166.916,54.325,159.988
C09806=1016.857,123.721,381.340,166.913,54.334,159.989
C09807=1016.852,123.471,381.359,166.909,54.344,159.990
C09808=1016.847,123.190,381.379,166.907,54.355,159.992
C09809=1016.841,122.909,381.400,166.903,54.365,159.993
C09810=1016.835,122.627,381.421,166.900,54.375,159.994
C09811=1016.830,122.346,381.442,166.897,54.386,159.996
C09812=1016.826,122.096,381.460,166.893,54.396,159.997
C09813=1016.821,121.847,381.478,166.890,54.405,159.998
C09814=1016.816,121.598,381.497,166.887,54.414,159.999
C09815=1016.811,121.349,381.515,166.885,54.424,160.001
C09816=1016.806,121.099,381.534,166.882,54.433,160.002
C09817=1016.801,120.850,381.552,166.878,54.442,160.003
C09818=1016.797,120.601,381.570,166.875,54.452,160.004
C09819=1016.792,120.352,381.589,166.873,54.461,160.005
C09820=1016.787,120.103,381.607,166.870,54.470,160.006
C09821=1016.782,119.853,381.625,166.866,54.480,160.008
C09822=1016.777,119.604,381.643,166.864,54.489,160.009
C09823=1016.772,119.355,381.662,166.861,54.498,160.010
C09824=1016.768,119.105,381.680,166.858,54.508,160.011
C09825=1016.763,118.857,381.699,166.855,54.517,160.012
C09826=1016.758,118.607,381.717,166.851,54.526,160.013
C09827=1016.753,118.358,381.735,166.848,54.535,160.015
C09828=1016.748,118.109,381.753,166.846,54.545,160.016
C09829=1016.743,117.859,381.771,166.843,54.554,160.017
C09830=1016.739,117.610,381.789,166.840,54.564,160.019
C09831=1016.734,117.360,381.808,166.837,54.573,160.020
C09832=1016.729,117.111,381.826,166.834,54.582,160.021
C09833=1016.724,116.862,381.844,166.831,54.591,160.022
C09834=1016.719,116.613,381.863,166.828,54.601,160.023
C09835=1016.714,116.364,381.881,166.825,54.610,160.024
C09836=1016.710,116.114,381.899,166.823,54.619,160.026
C09837=1016.705,115.865,381.917,166.820,54.629,160.027
C09838=1016.700,115.616,381.935,166.816,54.638,160.028
C09839=1016.695,115.366,381.954,166.814,54.648,160.029
C09840=1016.691,115.117,381.972,166.811,54.657,160.030
C09841=1016.687,114.867,381.990,166.808,54.666,160.032
C09842=1016.682,114.618,382.009,166.805,54.675,160.033
C09843=1016.677,114.369,382.027,166.802,54.684,160.034
C09844=1016.672,114.119,382.045,166.800,54.693,160.035
C09845=1016.667,113.870,382.063,166.796,54.703,160.036
C09846=1016.663,113.620,382.081,166.793,54.712,160.038
C09847=1016.658,113.371,382.099,166.790,54.721,160.039
C09848=1016.654,113.122,382.117,166.788,54.731,160.040
C09849=1016.649,112.873,382.135,166.785,54.740,160.041
C09850=1016.644,112.624,382.154,166.782,54.749,160.042
C09851=1016.639,112.374,382.172,166.779,54.758,160.044
C09852=1016.635,112.125,382.190,166.776,54.767,160.045
C09853=1016.630,111.876,382.208,166.774,54.777,160.046
C09854=1016.624,111.627,382.226,166.770,54.787,160.047
C09855=1016.620,111.377,382.243,166.768,54.796,160.049
C09856=1016.615,111.127,382.261,166.765,54.805,160.050
C09857=1016.610,110.878,382.279,166.762,54.814,160.051
C09858=1016.605,110.629,382.297,166.759,54.824,160.052
C09859=1016.600,110.380,382.315,166.756,54.833,160.053
C09860=1016.596,110.130,382.332,166.753,54.843,160.055
C09861=1016.591,109.881,382.350,166.751,54.852,160.056
C09862=1016.586,109.632,382.368,166.748,54.862,160.057
C09863=1016.581,109.383,382.386,166.745,54.871,160.058
C09864=1016.576,109.133,382.403,166.741,54.880,160.059
C09865=1016.571,108.884,382.421,166.739,54.890,160.061
C09866=1016.566,108.634,382.439,166.736,54.900,160.062
C09867=1016.561,108.385,382.456,166.734,54.909,160.063
C09868=1016.557,108.136,382.474,166.730,54.918,160.064
C09869=1016.551,107.887,382.491,166.728,54.928,160.066
C09870=1016.547,107.637,382.509,166.725,54.938,160.067
C09871=1016.541,107.388,382.526,166.722,54.947,160.068
C09872=1016.536,107.106,382.546,166.719,54.957,160.070
C09873=1016.530,106.825,382.566,166.715,54.969,160.071
C09874=1016.525,106.543,382.586,166.712,54.979,160.072
C09875=1016.519,106.263,382.605,166.709,54.990,160.074
C09876=1016.515,106.013,382.623,166.706,54.999,160.075
C09877=1016.510,105.763,382.641,166.704,55.008,160.076
C09878=1016.505,105.514,382.658,166.701,55.018,160.077
C09879=1016.500,105.265,382.677,166.697,55.027,160.079
C09880=1016.495,105.016,382.693,166.695,55.036,160.080
C09881=1016.490,104.767,382.711,166.692,55.046,160.081
C09882=1016.485,104.517,382.728,166.690,55.056,160.082
C09883=1016.480,104.268,382.746,166.687,55.065,160.084
C09884=1016.475,104.018,382.763,166.684,55.074,160.085
C09885=1016.471,103.769,382.781,166.681,55.084,160.086
C09886=1016.466,103.520,382.798,166.678,55.093,160.087
C09887=1016.461,103.270,382.816,166.676,55.103,160.089
C09888=1016.456,103.021,382.833,166.673,55.112,160.090
C09889=1016.451,102.771,382.851,166.670,55.121,160.091
C09890=1016.446,102.523,382.868,166.668,55.131,160.092
C09891=1016.442,102.273,382.886,166.664,55.140,160.093
C09892=1016.437,102.024,382.904,166.661,55.150,160.095
C09893=1016.432,101.774,382.921,166.659,55.159,160.096
C09894=1016.427,101.525,382.938,166.656,55.168,160.097
C09895=1016.422,101.276,382.955,166.653,55.177,160.098
C09896=1016.417,101.026,382.973,166.651,55.187,160.100
C09897=1016.412,100.777,382.990,166.648,55.197,160.101
C09898=1016.408,100.528,383.008,166.645,55.206,160.102
C09899=1016.403,100.278,383.025,166.642,55.216,160.103
C09900=1016.398,100.028,383.042,166.639,55.225,160.104
C09901=1016.393,99.779,383.060,166.637,55.234,160.106
C09902=1016.389,99.530,383.077,166.634,55.243,160.107
C09903=1016.383,99.281,383.095,166.631,55.253,160.108
C09904=1016.379,99.031,383.112,166.629,55.262,160.109
C09905=1016.374,98.782,383.128,166.626,55.271,160.111
C09906=1016.369,98.533,383.146,166.622,55.281,160.112
C09907=1016.364,98.283,383.163,166.620,55.291,160.113
C09908=1016.359,98.033,383.180,166.618,55.300,160.114
C09909=1016.354,97.785,383.198,166.615,55.309,160.116
C09910=1016.349,97.535,383.214,166.612,55.319,160.117
C09911=1016.345,97.285,383.232,166.609,55.329,160.118
C09912=1016.340,97.036,383.248,166.607,55.338,160.119
C09913=1016.334,96.787,383.266,166.604,55.348,160.121
C09914=1016.329,96.538,383.283,166.601,55.357,160.122
C09915=1016.325,96.288,383.300,166.599,55.366,160.123
C09916=1016.320,96.039,383.317,166.595,55.376,160.124
C09917=1016.315,95.789,383.334,166.593,55.386,160.126
C09918=1016.309,95.540,383.351,166.590,55.395,160.127
C09919=1016.305,95.291,383.368,166.588,55.405,160.128
C09920=1016.300,95.041,383.385,166.585,55.414,160.129
C09921=1016.295,94.791,383.402,166.582,55.423,160.131
C09922=1016.291,94.543,383.418,166.579,55.433,160.132
C09923=1016.285,94.293,383.436,166.576,55.442,160.133
C09924=1016.281,94.044,383.453,166.574,55.452,160.134
C09925=1016.276,93.795,383.470,166.571,55.461,160.136
C09926=1016.271,93.545,383.487,166.569,55.471,160.137
C09927=1016.266,93.296,383.503,166.566,55.480,160.138
C09928=1016.261,93.046,383.520,166.564,55.489,160.139
C09929=1016.256,92.797,383.538,166.560,55.499,160.140
C09930=1016.251,92.548,383.555,166.557,55.508,160.142
C09931=1016.246,92.298,383.572,166.555,55.518,160.143
C09932=1016.241,92.049,383.588,166.552,55.527,160.144
C09933=1016.237,91.799,383.605,166.550,55.536,160.145
C09934=1016.232,91.550,383.622,166.547,55.546,160.147
C09935=1016.227,91.301,383.639,166.544,55.555,160.148
C09936=1016.221,91.019,383.658,166.542,55.566,160.149
C09937=1016.216,90.738,383.677,166.539,55.577,160.151
C09938=1016.210,90.457,383.696,166.536,55.587,160.152
C09939=1016.205,90.176,383.715,166.533,55.597,160.153
C09940=1016.201,89.927,383.732,166.530,55.607,160.155
C09941=1016.196,89.677,383.749,166.526,55.616,160.156
C09942=1016.191,89.428,383.766,166.524,55.626,160.157
C09943=1016.186,89.179,383.783,166.521,55.635,160.158
C09944=1016.181,88.929,383.799,166.519,55.644,160.159
C09945=1016.177,88.680,383.817,166.516,55.654,160.161
C09946=1016.171,88.430,383.833,166.514,55.663,160.162
C09947=1016.166,88.181,383.850,166.512,55.673,160.163
C09948=1016.161,87.932,383.866,166.509,55.683,160.165
C09949=1016.156,87.682,383.883,166.505,55.692,160.166
C09950=1016.151,87.433,383.899,166.503,55.702,160.167
C09951=1016.146,87.183,383.916,166.500,55.711,160.168
C09952=1016.142,86.934,383.932,166.498,55.720,160.169
C09953=1016.137,86.684,383.949,166.496,55.730,160.171
C09954=1016.132,86.435,383.965,166.492,55.740,160.172
C09955=1016.127,86.186,383.982,166.490,55.749,160.173
C09956=1016.122,85.936,383.999,166.487,55.759,160.175
C09957=1016.116,85.687,384.014,166.484,55.768,160.176
C09958=1016.111,85.437,384.031,166.482,55.777,160.177
C09959=1016.107,85.188,384.048,166.479,55.787,160.178
C09960=1016.101,84.938,384.065,166.476,55.797,160.179
C09961=1016.097,84.689,384.081,166.474,55.807,160.181
C09962=1016.092,84.440,384.098,166.471,55.816,160.182
C09963=1016.087,84.190,384.114,166.469,55.825,160.183
C09964=1016.082,83.940,384.130,166.466,55.835,160.185
C09965=1016.077,83.692,384.147,166.464,55.844,160.186
C09966=1016.072,83.442,384.164,166.461,55.853,160.187
C09967=1016.067,83.193,384.179,166.458,55.863,160.188
C09968=1016.062,82.943,384.196,166.455,55.873,160.189
C09969=1016.057,82.694,384.212,166.453,55.882,160.191
C09970=1016.052,82.444,384.229,166.450,55.891,160.192
C09971=1016.048,82.195,384.246,166.448,55.901,160.193
C09972=1016.043,81.945,384.262,166.445,55.910,160.195
C09973=1016.038,81.696,384.278,166.443,55.919,160.196
C09974=1016.033,81.447,384.295,166.440,55.929,160.197
C09975=1016.029,81.197,384.311,166.438,55.938,160.198
C09976=1016.023,80.948,384.327,166.434,55.948,160.199
C09977=1016.018,80.699,384.344,166.432,55.957,160.201
C09978=1016.013,80.450,384.360,166.429,55.967,160.202
C09979=1016.008,80.199,384.376,166.427,55.976,160.203
C09980=1016.004,79.950,384.393,166.424,55.985,160.204
C09981=1015.999,79.701,384.410,166.422,55.995,160.206
C09982=1015.994,79.451,384.425,166.419,56.004,160.207
C09983=1015.990,79.202,384.442,166.417,56.014,160.208
C09984=1015.984,78.953,384.459,166.414,56.023,160.209
C09985=1015.980,78.704,384.475,166.412,56.032,160.211
C09986=1015.974,78.454,384.491,166.409,56.042,160.212
C09987=1015.970,78.205,384.507,166.407,56.051,160.213
C09988=1015.964,77.955,384.524,166.404,56.060,160.214
C09989=1015.960,77.705,384.540,166.401,56.069,160.215
C09990=1015.955,77.456,384.556,166.399,56.079,160.217
C09991=1015.951,77.206,384.572,166.396,56.088,160.218
C09992=1015.946,76.957,384.589,166.394,56.097,160.219
C09993=1015.940,76.708,384.605,166.390,56.107,160.220
C09994=1015.936,76.458,384.621,166.388,56.117,160.222
C09995=1015.931,76.209,384.637,166.386,56.126,160.223
C09996=1015.926,75.959,384.654,166.383,56.135,160.224
//INST
///DATE 2021/06/25 14:50
///ATTR SC,RW,RJ
////FRAME ROBOT
///GROUP1 RB1
NOP
MOVL C00000 V=800.0 PL=0
MOVL C00001 V=800.0 PL=0
MOVL C00002 V=800.0 PL=0
MOVL C00003 V=800.0 PL=0
MOVL C00004 V=800.0 PL=0
MOVL C00005 V=800.0 PL=0
MOVL C00006 V=800.0 PL=0
MOVL C00007 V=800.0 PL=0
MOVL C00008 V=800.0 PL=0
MOVL C00009 V=800.0 PL=0
MOVL C00010 V=800.0 PL=0
MOVL C00011 V=800.0 PL=0
MOVL C00012 V=800.0 PL=0
MOVL C00013 V=800.0 PL=0
MOVL C00014 V=800.0 PL=0
MOVL C00015 V=800.0 PL=0
MOVL C00016 V=800.0 PL=0
MOVL C00017 V=800.0 PL=0
MOVL C00018 V=800.0 PL=0
MOVL C00019 V=800.0 PL=0
MOVL C00020 V=800.0 PL=0
MOVL C00021 V=800.0 PL=0
MOVL C00022 V=800.0 PL=0
MOVL C00023 V=800.0 PL=0
MOVL C00024 V=800.0 PL=0
MOVL C00025 V=800.0 PL=0
MOVL C00026 V=800.0 PL=0
MOVL C00027 V=800.0 PL=0
MOVL C00028 V=800.0 PL=0
MOVL C00029 V=800.0 PL=0
MOVL C00030 V=800.0 PL=0
MOVL C00031 V=800.0 PL=0
MOVL C00032 V=800.0 PL=0
MOVL C00033 V=800.0 PL=0
MOVL C00034 V=800.0 PL=0
MOVL C00035 V=800.0 PL=0
MOVL C00036 V=800.0 PL=0
MOVL C00037 V=800.0 PL=0
MOVL C00038 V=800.0 PL=0
MOVL C00039 V=800.0 PL=0
MOVL C00040 V=800.0 PL=0
MOVL C00041 V=800.0 PL=0
MOVL C00042 V=800.0 PL=0
MOVL C00043 V=800.0 PL=0
MOVL C00044 V=800.0 PL=0
MOVL C00045 V=800.0 PL=0
MOVL C00046 V=800.0 PL=0
MOVL C00047 V=800.0 PL=0
MOVL C00048 V=800.0 PL=0
MOVL C00049 V=800.0 PL=0
MOVL C00050 V=800.0 PL=0
MOVL C00051 V=800.0 PL=0
MOVL C00052 V=800.0 PL=0
MOVL C00053 V=800.0 PL=0
MOVL C00054 V=800.0 PL=0
MOVL C00055 V=800.0 PL=0
MOVL C00056 V=800.0 PL=0
MOVL C00057 V=800.0 PL=0
MOVL C00058 V=800.0 PL=0
MOVL C00059 V=800.0 PL=0
MOVL C00060 V=800.0 PL=0
MOVL C00061 V=800.0 PL=0
MOVL C00062 V=800.0 PL=0
MOVL C00063 V=800.0 PL=0
MOVL C00064 V=800.0 PL=0
MOVL C00065 V=800.0 PL=0
MOVL C00066 V=800.0 PL=0
MOVL C00067 V=800.0 PL=0
MOVL C00068 V=800.0 PL=0
MOVL C00069 V=800.0 PL=0
MOVL C00070 V=800.0 PL=0
MOVL C00071 V=800.0 PL=0
MOVL C00072 V=800.0 PL=0
MOVL C00073 V=800.0 PL=0
MOVL C00074 V=800.0 PL=0
MOVL C00075 V=800.0 PL=0
MOVL C00076 V=800.0 PL=0
MOVL C00077 V=800.0 PL=0
MOVL C00078 V=800.0 PL=0
MOVL C00079 V=800.0 PL=0
MOVL C00080 V=800.0 PL=0
MOVL C00081 V=800.0 PL=0
MOVL C00082 V=800.0 PL=0
MOVL C00083 V=800.0 PL=0
MOVL C00084 V=800.0 PL=0
MOVL C00085 V=800.0 PL=0
MOVL C00086 V=800.0 PL=0
MOVL C00087 V=800.0 PL=0
MOVL C00088 V=800.0 PL=0
MOVL C00089 V=800.0 PL=0
MOVL C00090 V=800.0 PL=0
MOVL C00091 V=800.0 PL=0
MOVL C00092 V=800.0 PL=0
MOVL C00093 V=800.0 PL=0
MOVL C00094 V=800.0 PL=0
MOVL C00095 V=800.0 PL=0
MOVL C00096 V=800.0 PL=0
MOVL C00097 V=800.0 PL=0
MOVL C00098 V=800.0 PL=0
MOVL C00099 V=800.0 PL=0
MOVL C00100 V=800.0 PL=0
MOVL C00101 V=800.0 PL=0
MOVL C00102 V=800.0 PL=0
MOVL C00103 V=800.0 PL=0
MOVL C00104 V=800.0 PL=0
MOVL C00105 V=800.0 PL=0
MOVL C00106 V=800.0 PL=0
MOVL C00107 V=800.0 PL=0
MOVL C00108 V=800.0 PL=0
MOVL C00109 V=800.0 PL=0
MOVL C00110 V=800.0 PL=0
MOVL C00111 V=800.0 PL=0
MOVL C00112 V=800.0 PL=0
MOVL C00113 V=800.0 PL=0
MOVL C00114 V=800.0 PL=0
MOVL C00115 V=800.0 PL=0
MOVL C00116 V=800.0 PL=0
MOVL C00117 V=800.0 PL=0
MOVL C00118 V=800.0 PL=0
MOVL C00119 V=800.0 PL=0
MOVL C00120 V=800.0 PL=0
MOVL C00121 V=800.0 PL=0
MOVL C00122 V=800.0 PL=0
MOVL C00123 V=800.0 PL=0
MOVL C00124 V=800.0 PL=0
MOVL C00125 V=800.0 PL=0
MOVL C00126 V=800.0 PL=0
MOVL C00127 V=800.0 PL=0
MOVL C00128 V=800.0 PL=0
MOVL C00129 V=800.0 PL=0
MOVL C00130 V=800.0 PL=0
MOVL C00131 V=800.0 PL=0
MOVL C00132 V=800.0 PL=0
MOVL C00133 V=800.0 PL=0
MOVL C00134 V=800.0 PL=0
MOVL C00135 V=800.0 PL=0
MOVL C00136 V=800.0 PL=0
MOVL C00137 V=800.0 PL=0
MOVL C00138 V=800.0 PL=0
MOVL C00139 V=800.0 PL=0
MOVL C00140 V=800.0 PL=0
MOVL C00141 V=800.0 PL=0
MOVL C00142 V=800.0 PL=0
MOVL C00143 V=800.0 PL=0
MOVL C00144 V=800.0 PL=0
MOVL C00145 V=800.0 PL=0
MOVL C00146 V=800.0 PL=0
MOVL C00147 V=800.0 PL=0
MOVL C00148 V=800.0 PL=0
MOVL C00149 V=800.0 PL=0
MOVL C00150 V=800.0 PL=0
MOVL C00151 V=800.0 PL=0
MOVL C00152 V=800.0 PL=0
MOVL C00153 V=800.0 PL=0
MOVL C00154 V=800.0 PL=0
MOVL C00155 V=800.0 PL=0
MOVL C00156 V=800.0 PL=0
MOVL C00157 V=800.0 PL=0
MOVL C00158 V=800.0 PL=0
MOVL C00159 V=800.0 PL=0
MOVL C00160 V=800.0 PL=0
MOVL C00161 V=800.0 PL=0
MOVL C00162 V=800.0 PL=0
MOVL C00163 V=800.0 PL=0
MOVL C00164 V=800.0 PL=0
MOVL C00165 V=800.0 PL=0
MOVL C00166 V=800.0 PL=0
MOVL C00167 V=800.0 PL=0
MOVL C00168 V=800.0 PL=0
MOVL C00169 V=800.0 PL=0
MOVL C00170 V=800.0 PL=0
MOVL C00171 V=800.0 PL=0
MOVL C00172 V=800.0 PL=0
MOVL C00173 V=800.0 PL=0
MOVL C00174 V=800.0 PL=0
MOVL C00175 V=800.0 PL=0
MOVL C00176 V=800.0 PL=0
MOVL C00177 V=800.0 PL=0
MOVL C00178 V=800.0 PL=0
MOVL C00179 V=800.0 PL=0
MOVL C00180 V=800.0 PL=0
MOVL C00181 V=800.0 PL=0
MOVL C00182 V=800.0 PL=0
MOVL C00183 V=800.0 PL=0
MOVL C00184 V=800.0 PL=0
MOVL C00185 V=800.0 PL=0
MOVL C00186 V=800.0 PL=0
MOVL C00187 V=800.0 PL=0
MOVL C00188 V=800.0 PL=0
MOVL C00189 V=800.0 PL=0
MOVL C00190 V=800.0 PL=0
MOVL C00191 V=800.0 PL=0
MOVL C00192 V=800.0 PL=0
MOVL C00193 V=800.0 PL=0
MOVL C00194 V=800.0 PL=0
MOVL C00195 V=800.0 PL=0
MOVL C00196 V=800.0 PL=0
MOVL C00197 V=800.0 PL=0
MOVL C00198 V=800.0 PL=0
MOVL C00199 V=800.0 PL=0
MOVL C00200 V=800.0 PL=0
MOVL C00201 V=800.0 PL=0
MOVL C00202 V=800.0 PL=0
MOVL C00203 V=800.0 PL=0
MOVL C00204 V=800.0 PL=0
MOVL C00205 V=800.0 PL=0
MOVL C00206 V=800.0 PL=0
MOVL C00207 V=800.0 PL=0
MOVL C00208 V=800.0 PL=0
MOVL C00209 V=800.0 PL=0
MOVL C00210 V=800.0 PL=0
MOVL C00211 V=800.0 PL=0
MOVL C00212 V=800.0 PL=0
MOVL C00213 V=800.0 PL=0
MOVL C00214 V=800.0 PL=0
MOVL C00215 V=800.0 PL=0
MOVL C00216 V=800.0 PL=0
MOVL C00217 V=800.0 PL=0
MOVL C00218 V=800.0 PL=0
MOVL C00219 V=800.0 PL=0
MOVL C00220 V=800.0 PL=0
MOVL C00221 V=800.0 PL=0
MOVL C00222 V=800.0 PL=0
MOVL C00223 V=800.0 PL=0
MOVL C00224 V=800.0 PL=0
MOVL C00225 V=800.0 PL=0
MOVL C00226 V=800.0 PL=0
MOVL C00227 V=800.0 PL=0
MOVL C00228 V=800.0 PL=0
MOVL C00229 V=800.0 PL=0
MOVL C00230 V=800.0 PL=0
MOVL C00231 V=800.0 PL=0
MOVL C00232 V=800.0 PL=0
MOVL C00233 V=800.0 PL=0
MOVL C00234 V=800.0 PL=0
MOVL C00235 V=800.0 PL=0
MOVL C00236 V=800.0 PL=0
MOVL C00237 V=800.0 PL=0
MOVL C00238 V=800.0 PL=0
MOVL C00239 V=800.0 PL=0
MOVL C00240 V=800.0 PL=0
MOVL C00241 V=800.0 PL=0
MOVL C00242 V=800.0 PL=0
MOVL C00243 V=800.0 PL=0
MOVL C00244 V=800.0 PL=0
MOVL C00245 V=800.0 PL=0
MOVL C00246 V=800.0 PL=0
MOVL C00247 V=800.0 PL=0
MOVL C00248 V=800.0 PL=0
MOVL C00249 V=800.0 PL=0
MOVL C00250 V=800.0 PL=0
MOVL C00251 V=800.0 PL=0
MOVL C00252 V=800.0 PL=0
MOVL C00253 V=800.0 PL=0
MOVL C00254 V=800.0 PL=0
MOVL C00255 V=800.0 PL=0
MOVL C00256 V=800.0 PL=0
MOVL C00257 V=800.0 PL=0
MOVL C00258 V=800.0 PL=0
MOVL C00259 V=800.0 PL=0
MOVL C00260 V=800.0 PL=0
MOVL C00261 V=800.0 PL=0
MOVL C00262 V=800.0 PL=0
MOVL C00263 V=800.0 PL=0
MOVL C00264 V=800.0 PL=0
MOVL C00265 V=800.0 PL=0
MOVL C00266 V=800.0 PL=0
MOVL C00267 V=800.0 PL=0
MOVL C00268 V=800.0 PL=0
MOVL C00269 V=800.0 PL=0
MOVL C00270 V=800.0 PL=0
MOVL C00271 V=800.0 PL=0
MOVL C00272 V=800.0 PL=0
MOVL C00273 V=800.0 PL=0
MOVL C00274 V=800.0 PL=0
MOVL C00275 V=800.0 PL=0
MOVL C00276 V=800.0 PL=0
MOVL C00277 V=800.0 PL=0
MOVL C00278 V=800.0 PL=0
MOVL C00279 V=800.0 PL=0
MOVL C00280 V=800.0 PL=0
MOVL C00281 V=800.0 PL=0
MOVL C00282 V=800.0 PL=0
MOVL C00283 V=800.0 PL=0
MOVL C00284 V=800.0 PL=0
MOVL C00285 V=800.0 PL=0
MOVL C00286 V=800.0 PL=0
MOVL C00287 V=800.0 PL=0
MOVL C00288 V=800.0 PL=0
MOVL C00289 V=800.0 PL=0
MOVL C00290 V=800.0 PL=0
MOVL C00291 V=800.0 PL=0
MOVL C00292 V=800.0 PL=0
MOVL C00293 V=800.0 PL=0
MOVL C00294 V=800.0 PL=0
MOVL C00295 V=800.0 PL=0
MOVL C00296 V=800.0 PL=0
MOVL C00297 V=800.0 PL=0
MOVL C00298 V=800.0 PL=0
MOVL C00299 V=800.0 PL=0
MOVL C00300 V=800.0 PL=0
MOVL C00301 V=800.0 PL=0
MOVL C00302 V=800.0 PL=0
MOVL C00303 V=800.0 PL=0
MOVL C00304 V=800.0 PL=0
MOVL C00305 V=800.0 PL=0
MOVL C00306 V=800.0 PL=0
MOVL C00307 V=800.0 PL=0
MOVL C00308 V=800.0 PL=0
MOVL C00309 V=800.0 PL=0
MOVL C00310 V=800.0 PL=0
MOVL C00311 V=800.0 PL=0
MOVL C00312 V=800.0 PL=0
MOVL C00313 V=800.0 PL=0
MOVL C00314 V=800.0 PL=0
MOVL C00315 V=800.0 PL=0
MOVL C00316 V=800.0 PL=0
MOVL C00317 V=800.0 PL=0
MOVL C00318 V=800.0 PL=0
MOVL C00319 V=800.0 PL=0
MOVL C00320 V=800.0 PL=0
MOVL C00321 V=800.0 PL=0
MOVL C00322 V=800.0 PL=0
MOVL C00323 V=800.0 PL=0
MOVL C00324 V=800.0 PL=0
MOVL C00325 V=800.0 PL=0
MOVL C00326 V=800.0 PL=0
MOVL C00327 V=800.0 PL=0
MOVL C00328 V=800.0 PL=0
MOVL C00329 V=800.0 PL=0
MOVL C00330 V=800.0 PL=0
MOVL C00331 V=800.0 PL=0
MOVL C00332 V=800.0 PL=0
MOVL C00333 V=800.0 PL=0
MOVL C00334 V=800.0 PL=0
MOVL C00335 V=800.0 PL=0
MOVL C00336 V=800.0 PL=0
MOVL C00337 V=800.0 PL=0
MOVL C00338 V=800.0 PL=0
MOVL C00339 V=800.0 PL=0
MOVL C00340 V=800.0 PL=0
MOVL C00341 V=800.0 PL=0
MOVL C00342 V=800.0 PL=0
MOVL C00343 V=800.0 PL=0
MOVL C00344 V=800.0 PL=0
MOVL C00345 V=800.0 PL=0
MOVL C00346 V=800.0 PL=0
MOVL C00347 V=800.0 PL=0
MOVL C00348 V=800.0 PL=0
MOVL C00349 V=800.0 PL=0
MOVL C00350 V=800.0 PL=0
MOVL C00351 V=800.0 PL=0
MOVL C00352 V=800.0 PL=0
MOVL C00353 V=800.0 PL=0
MOVL C00354 V=800.0 PL=0
MOVL C00355 V=800.0 PL=0
MOVL C00356 V=800.0 PL=0
MOVL C00357 V=800.0 PL=0
MOVL C00358 V=800.0 PL=0
MOVL C00359 V=800.0 PL=0
MOVL C00360 V=800.0 PL=0
MOVL C00361 V=800.0 PL=0
MOVL C00362 V=800.0 PL=0
MOVL C00363 V=800.0 PL=0
MOVL C00364 V=800.0 PL=0
MOVL C00365 V=800.0 PL=0
MOVL C00366 V=800.0 PL=0
MOVL C00367 V=800.0 PL=0
MOVL C00368 V=800.0 PL=0
MOVL C00369 V=800.0 PL=0
MOVL C00370 V=800.0 PL=0
MOVL C00371 V=800.0 PL=0
MOVL C00372 V=800.0 PL=0
MOVL C00373 V=800.0 PL=0
MOVL C00374 V=800.0 PL=0
MOVL C00375 V=800.0 PL=0
MOVL C00376 V=800.0 PL=0
MOVL C00377 V=800.0 PL=0
MOVL C00378 V=800.0 PL=0
MOVL C00379 V=800.0 PL=0
MOVL C00380 V=800.0 PL=0
MOVL C00381 V=800.0 PL=0
MOVL C00382 V=800.0 PL=0
MOVL C00383 V=800.0 PL=0
MOVL C00384 V=800.0 PL=0
MOVL C00385 V=800.0 PL=0
MOVL C00386 V=800.0 PL=0
MOVL C00387 V=800.0 PL=0
MOVL C00388 V=800.0 PL=0
MOVL C00389 V=800.0 PL=0
MOVL C00390 V=800.0 PL=0
MOVL C00391 V=800.0 PL=0
MOVL C00392 V=800.0 PL=0
MOVL C00393 V=800.0 PL=0
MOVL C00394 V=800.0 PL=0
MOVL C00395 V=800.0 PL=0
MOVL C00396 V=800.0 PL=0
MOVL C00397 V=800.0 PL=0
MOVL C00398 V=800.0 PL=0
MOVL C00399 V=800.0 PL=0
MOVL C00400 V=800.0 PL=0
MOVL C00401 V=800.0 PL=0
MOVL C00402 V=800.0 PL=0
MOVL C00403 V=800.0 PL=0
MOVL C00404 V=800.0 PL=0
MOVL C00405 V=800.0 PL=0
MOVL C00406 V=800.0 PL=0
MOVL C00407 V=800.0 PL=0
MOVL C00408 V=800.0 PL=0
MOVL C00409 V=800.0 PL=0
MOVL C00410 V=800.0 PL=0
MOVL C00411 V=800.0 PL=0
MOVL C00412 V=800.0 PL=0
MOVL C00413 V=800.0 PL=0
MOVL C00414 V=800.0 PL=0
MOVL C00415 V=800.0 PL=0
MOVL C00416 V=800.0 PL=0
MOVL C00417 V=800.0 PL=0
MOVL C00418 V=800.0 PL=0
MOVL C00419 V=800.0 PL=0
MOVL C00420 V=800.0 PL=0
MOVL C00421 V=800.0 PL=0
MOVL C00422 V=800.0 PL=0
MOVL C00423 V=800.0 PL=0
MOVL C00424 V=800.0 PL=0
MOVL C00425 V=800.0 PL=0
MOVL C00426 V=800.0 PL=0
MOVL C00427 V=800.0 PL=0
MOVL C00428 V=800.0 PL=0
MOVL C00429 V=800.0 PL=0
MOVL C00430 V=800.0 PL=0
MOVL C00431 V=800.0 PL=0
MOVL C00432 V=800.0 PL=0
MOVL C00433 V=800.0 PL=0
MOVL C00434 V=800.0 PL=0
MOVL C00435 V=800.0 PL=0
MOVL C00436 V=800.0 PL=0
MOVL C00437 V=800.0 PL=0
MOVL C00438 V=800.0 PL=0
MOVL C00439 V=800.0 PL=0
MOVL C00440 V=800.0 PL=0
MOVL C00441 V=800.0 PL=0
MOVL C00442 V=800.0 PL=0
MOVL C00443 V=800.0 PL=0
MOVL C00444 V=800.0 PL=0
MOVL C00445 V=800.0 PL=0
MOVL C00446 V=800.0 PL=0
MOVL C00447 V=800.0 PL=0
MOVL C00448 V=800.0 PL=0
MOVL C00449 V=800.0 PL=0
MOVL C00450 V=800.0 PL=0
MOVL C00451 V=800.0 PL=0
MOVL C00452 V=800.0 PL=0
MOVL C00453 V=800.0 PL=0
MOVL C00454 V=800.0 PL=0
MOVL C00455 V=800.0 PL=0
MOVL C00456 V=800.0 PL=0
MOVL C00457 V=800.0 PL=0
MOVL C00458 V=800.0 PL=0
MOVL C00459 V=800.0 PL=0
MOVL C00460 V=800.0 PL=0
MOVL C00461 V=800.0 PL=0
MOVL C00462 V=800.0 PL=0
MOVL C00463 V=800.0 PL=0
MOVL C00464 V=800.0 PL=0
MOVL C00465 V=800.0 PL=0
MOVL C00466 V=800.0 PL=0
MOVL C00467 V=800.0 PL=0
MOVL C00468 V=800.0 PL=0
MOVL C00469 V=800.0 PL=0
MOVL C00470 V=800.0 PL=0
MOVL C00471 V=800.0 PL=0
MOVL C00472 V=800.0 PL=0
MOVL C00473 V=800.0 PL=0
MOVL C00474 V=800.0 PL=0
MOVL C00475 V=800.0 PL=0
MOVL C00476 V=800.0 PL=0
MOVL C00477 V=800.0 PL=0
MOVL C00478 V=800.0 PL=0
MOVL C00479 V=800.0 PL=0
MOVL C00480 V=800.0 PL=0
MOVL C00481 V=800.0 PL=0
MOVL C00482 V=800.0 PL=0
MOVL C00483 V=800.0 PL=0
MOVL C00484 V=800.0 PL=0
MOVL C00485 V=800.0 PL=0
MOVL C00486 V=800.0 PL=0
MOVL C00487 V=800.0 PL=0
MOVL C00488 V=800.0 PL=0
MOVL C00489 V=800.0 PL=0
MOVL C00490 V=800.0 PL=0
MOVL C00491 V=800.0 PL=0
MOVL C00492 V=800.0 PL=0
MOVL C00493 V=800.0 PL=0
MOVL C00494 V=800.0 PL=0
MOVL C00495 V=800.0 PL=0
MOVL C00496 V=800.0 PL=0
MOVL C00497 V=800.0 PL=0
MOVL C00498 V=800.0 PL=0
MOVL C00499 V=800.0 PL=0
MOVL C00500 V=800.0 PL=0
MOVL C00501 V=800.0 PL=0
MOVL C00502 V=800.0 PL=0
MOVL C00503 V=800.0 PL=0
MOVL C00504 V=800.0 PL=0
MOVL C00505 V=800.0 PL=0
MOVL C00506 V=800.0 PL=0
MOVL C00507 V=800.0 PL=0
MOVL C00508 V=800.0 PL=0
MOVL C00509 V=800.0 PL=0
MOVL C00510 V=800.0 PL=0
MOVL C00511 V=800.0 PL=0
MOVL C00512 V=800.0 PL=0
MOVL C00513 V=800.0 PL=0
MOVL C00514 V=800.0 PL=0
MOVL C00515 V=800.0 PL=0
MOVL C00516 V=800.0 PL=0
MOVL C00517 V=800.0 PL=0
MOVL C00518 V=800.0 PL=0
MOVL C00519 V=800.0 PL=0
MOVL C00520 V=800.0 PL=0
MOVL C00521 V=800.0 PL=0
MOVL C00522 V=800.0 PL=0
MOVL C00523 V=800.0 PL=0
MOVL C00524 V=800.0 PL=0
MOVL C00525 V=800.0 PL=0
MOVL C00526 V=800.0 PL=0
MOVL C00527 V=800.0 PL=0
MOVL C00528 V=800.0 PL=0
MOVL C00529 V=800.0 PL=0
MOVL C00530 V=800.0 PL=0
MOVL C00531 V=800.0 PL=0
MOVL C00532 V=800.0 PL=0
MOVL C00533 V=800.0 PL=0
MOVL C00534 V=800.0 PL=0
MOVL C00535 V=800.0 PL=0
MOVL C00536 V=800.0 PL=0
MOVL C00537 V=800.0 PL=0
MOVL C00538 V=800.0 PL=0
MOVL C00539 V=800.0 PL=0
MOVL C00540 V=800.0 PL=0
MOVL C00541 V=800.0 PL=0
MOVL C00542 V=800.0 PL=0
MOVL C00543 V=800.0 PL=0
MOVL C00544 V=800.0 PL=0
MOVL C00545 V=800.0 PL=0
MOVL C00546 V=800.0 PL=0
MOVL C00547 V=800.0 PL=0
MOVL C00548 V=800.0 PL=0
MOVL C00549 V=800.0 PL=0
MOVL C00550 V=800.0 PL=0
MOVL C00551 V=800.0 PL=0
MOVL C00552 V=800.0 PL=0
MOVL C00553 V=800.0 PL=0
MOVL C00554 V=800.0 PL=0
MOVL C00555 V=800.0 PL=0
MOVL C00556 V=800.0 PL=0
MOVL C00557 V=800.0 PL=0
MOVL C00558 V=800.0 PL=0
MOVL C00559 V=800.0 PL=0
MOVL C00560 V=800.0 PL=0
MOVL C00561 V=800.0 PL=0
MOVL C00562 V=800.0 PL=0
MOVL C00563 V=800.0 PL=0
MOVL C00564 V=800.0 PL=0
MOVL C00565 V=800.0 PL=0
MOVL C00566 V=800.0 PL=0
MOVL C00567 V=800.0 PL=0
MOVL C00568 V=800.0 PL=0
MOVL C00569 V=800.0 PL=0
MOVL C00570 V=800.0 PL=0
MOVL C00571 V=800.0 PL=0
MOVL C00572 V=800.0 PL=0
MOVL C00573 V=800.0 PL=0
MOVL C00574 V=800.0 PL=0
MOVL C00575 V=800.0 PL=0
MOVL C00576 V=800.0 PL=0
MOVL C00577 V=800.0 PL=0
MOVL C00578 V=800.0 PL=0
MOVL C00579 V=800.0 PL=0
MOVL C00580 V=800.0 PL=0
MOVL C00581 V=800.0 PL=0
MOVL C00582 V=800.0 PL=0
MOVL C00583 V=800.0 PL=0
MOVL C00584 V=800.0 PL=0
MOVL C00585 V=800.0 PL=0
MOVL C00586 V=800.0 PL=0
MOVL C00587 V=800.0 PL=0
MOVL C00588 V=800.0 PL=0
MOVL C00589 V=800.0 PL=0
MOVL C00590 V=800.0 PL=0
MOVL C00591 V=800.0 PL=0
MOVL C00592 V=800.0 PL=0
MOVL C00593 V=800.0 PL=0
MOVL C00594 V=800.0 PL=0
MOVL C00595 V=800.0 PL=0
MOVL C00596 V=800.0 PL=0
MOVL C00597 V=800.0 PL=0
MOVL C00598 V=800.0 PL=0
MOVL C00599 V=800.0 PL=0
MOVL C00600 V=800.0 PL=0
MOVL C00601 V=800.0 PL=0
MOVL C00602 V=800.0 PL=0
MOVL C00603 V=800.0 PL=0
MOVL C00604 V=800.0 PL=0
MOVL C00605 V=800.0 PL=0
MOVL C00606 V=800.0 PL=0
MOVL C00607 V=800.0 PL=0
MOVL C00608 V=800.0 PL=0
MOVL C00609 V=800.0 PL=0
MOVL C00610 V=800.0 PL=0
MOVL C00611 V=800.0 PL=0
MOVL C00612 V=800.0 PL=0
MOVL C00613 V=800.0 PL=0
MOVL C00614 V=800.0 PL=0
MOVL C00615 V=800.0 PL=0
MOVL C00616 V=800.0 PL=0
MOVL C00617 V=800.0 PL=0
MOVL C00618 V=800.0 PL=0
MOVL C00619 V=800.0 PL=0
MOVL C00620 V=800.0 PL=0
MOVL C00621 V=800.0 PL=0
MOVL C00622 V=800.0 PL=0
MOVL C00623 V=800.0 PL=0
MOVL C00624 V=800.0 PL=0
MOVL C00625 V=800.0 PL=0
MOVL C00626 V=800.0 PL=0
MOVL C00627 V=800.0 PL=0
MOVL C00628 V=800.0 PL=0
MOVL C00629 V=800.0 PL=0
MOVL C00630 V=800.0 PL=0
MOVL C00631 V=800.0 PL=0
MOVL C00632 V=800.0 PL=0
MOVL C00633 V=800.0 PL=0
MOVL C00634 V=800.0 PL=0
MOVL C00635 V=800.0 PL=0
MOVL C00636 V=800.0 PL=0
MOVL C00637 V=800.0 PL=0
MOVL C00638 V=800.0 PL=0
MOVL C00639 V=800.0 PL=0
MOVL C00640 V=800.0 PL=0
MOVL C00641 V=800.0 PL=0
MOVL C00642 V=800.0 PL=0
MOVL C00643 V=800.0 PL=0
MOVL C00644 V=800.0 PL=0
MOVL C00645 V=800.0 PL=0
MOVL C00646 V=800.0 PL=0
MOVL C00647 V=800.0 PL=0
MOVL C00648 V=800.0 PL=0
MOVL C00649 V=800.0 PL=0
MOVL C00650 V=800.0 PL=0
MOVL C00651 V=800.0 PL=0
MOVL C00652 V=800.0 PL=0
MOVL C00653 V=800.0 PL=0
MOVL C00654 V=800.0 PL=0
MOVL C00655 V=800.0 PL=0
MOVL C00656 V=800.0 PL=0
MOVL C00657 V=800.0 PL=0
MOVL C00658 V=800.0 PL=0
MOVL C00659 V=800.0 PL=0
MOVL C00660 V=800.0 PL=0
MOVL C00661 V=800.0 PL=0
MOVL C00662 V=800.0 PL=0
MOVL C00663 V=800.0 PL=0
MOVL C00664 V=800.0 PL=0
MOVL C00665 V=800.0 PL=0
MOVL C00666 V=800.0 PL=0
MOVL C00667 V=800.0 PL=0
MOVL C00668 V=800.0 PL=0
MOVL C00669 V=800.0 PL=0
MOVL C00670 V=800.0 PL=0
MOVL C00671 V=800.0 PL=0
MOVL C00672 V=800.0 PL=0
MOVL C00673 V=800.0 PL=0
MOVL C00674 V=800.0 PL=0
MOVL C00675 V=800.0 PL=0
MOVL C00676 V=800.0 PL=0
MOVL C00677 V=800.0 PL=0
MOVL C00678 V=800.0 PL=0
MOVL C00679 V=800.0 PL=0
MOVL C00680 V=800.0 PL=0
MOVL C00681 V=800.0 PL=0
MOVL C00682 V=800.0 PL=0
MOVL C00683 V=800.0 PL=0
MOVL C00684 V=800.0 PL=0
MOVL C00685 V=800.0 PL=0
MOVL C00686 V=800.0 PL=0
MOVL C00687 V=800.0 PL=0
MOVL C00688 V=800.0 PL=0
MOVL C00689 V=800.0 PL=0
MOVL C00690 V=800.0 PL=0
MOVL C00691 V=800.0 PL=0
MOVL C00692 V=800.0 PL=0
MOVL C00693 V=800.0 PL=0
MOVL C00694 V=800.0 PL=0
MOVL C00695 V=800.0 PL=0
MOVL C00696 V=800.0 PL=0
MOVL C00697 V=800.0 PL=0
MOVL C00698 V=800.0 PL=0
MOVL C00699 V=800.0 PL=0
MOVL C00700 V=800.0 PL=0
MOVL C00701 V=800.0 PL=0
MOVL C00702 V=800.0 PL=0
MOVL C00703 V=800.0 PL=0
MOVL C00704 V=800.0 PL=0
MOVL C00705 V=800.0 PL=0
MOVL C00706 V=800.0 PL=0
MOVL C00707 V=800.0 PL=0
MOVL C00708 V=800.0 PL=0
MOVL C00709 V=800.0 PL=0
MOVL C00710 V=800.0 PL=0
MOVL C00711 V=800.0 PL=0
MOVL C00712 V=800.0 PL=0
MOVL C00713 V=800.0 PL=0
MOVL C00714 V=800.0 PL=0
MOVL C00715 V=800.0 PL=0
MOVL C00716 V=800.0 PL=0
MOVL C00717 V=800.0 PL=0
MOVL C00718 V=800.0 PL=0
MOVL C00719 V=800.0 PL=0
MOVL C00720 V=800.0 PL=0
MOVL C00721 V=800.0 PL=0
MOVL C00722 V=800.0 PL=0
MOVL C00723 V=800.0 PL=0
MOVL C00724 V=800.0 PL=0
MOVL C00725 V=800.0 PL=0
MOVL C00726 V=800.0 PL=0
MOVL C00727 V=800.0 PL=0
MOVL C00728 V=800.0 PL=0
MOVL C00729 V=800.0 PL=0
MOVL C00730 V=800.0 PL=0
MOVL C00731 V=800.0 PL=0
MOVL C00732 V=800.0 PL=0
MOVL C00733 V=800.0 PL=0
MOVL C00734 V=800.0 PL=0
MOVL C00735 V=800.0 PL=0
MOVL C00736 V=800.0 PL=0
MOVL C00737 V=800.0 PL=0
MOVL C00738 V=800.0 PL=0
MOVL C00739 V=800.0 PL=0
MOVL C00740 V=800.0 PL=0
MOVL C00741 V=800.0 PL=0
MOVL C00742 V=800.0 PL=0
MOVL C00743 V=800.0 PL=0
MOVL C00744 V=800.0 PL=0
MOVL C00745 V=800.0 PL=0
MOVL C00746 V=800.0 PL=0
MOVL C00747 V=800.0 PL=0
MOVL C00748 V=800.0 PL=0
MOVL C00749 V=800.0 PL=0
MOVL C00750 V=800.0 PL=0
MOVL C00751 V=800.0 PL=0
MOVL C00752 V=800.0 PL=0
MOVL C00753 V=800.0 PL=0
MOVL C00754 V=800.0 PL=0
MOVL C00755 V=800.0 PL=0
MOVL C00756 V=800.0 PL=0
MOVL C00757 V=800.0 PL=0
MOVL C00758 V=800.0 PL=0
MOVL C00759 V=800.0 PL=0
MOVL C00760 V=800.0 PL=0
MOVL C00761 V=800.0 PL=0
MOVL C00762 V=800.0 PL=0
MOVL C00763 V=800.0 PL=0
MOVL C00764 V=800.0 PL=0
MOVL C00765 V=800.0 PL=0
MOVL C00766 V=800.0 PL=0
MOVL C00767 V=800.0 PL=0
MOVL C00768 V=800.0 PL=0
MOVL C00769 V=800.0 PL=0
MOVL C00770 V=800.0 PL=0
MOVL C00771 V=800.0 PL=0
MOVL C00772 V=800.0 PL=0
MOVL C00773 V=800.0 PL=0
MOVL C00774 V=800.0 PL=0
MOVL C00775 V=800.0 PL=0
MOVL C00776 V=800.0 PL=0
MOVL C00777 V=800.0 PL=0
MOVL C00778 V=800.0 PL=0
MOVL C00779 V=800.0 PL=0
MOVL C00780 V=800.0 PL=0
MOVL C00781 V=800.0 PL=0
MOVL C00782 V=800.0 PL=0
MOVL C00783 V=800.0 PL=0
MOVL C00784 V=800.0 PL=0
MOVL C00785 V=800.0 PL=0
MOVL C00786 V=800.0 PL=0
MOVL C00787 V=800.0 PL=0
MOVL C00788 V=800.0 PL=0
MOVL C00789 V=800.0 PL=0
MOVL C00790 V=800.0 PL=0
MOVL C00791 V=800.0 PL=0
MOVL C00792 V=800.0 PL=0
MOVL C00793 V=800.0 PL=0
MOVL C00794 V=800.0 PL=0
MOVL C00795 V=800.0 PL=0
MOVL C00796 V=800.0 PL=0
MOVL C00797 V=800.0 PL=0
MOVL C00798 V=800.0 PL=0
MOVL C00799 V=800.0 PL=0
MOVL C00800 V=800.0 PL=0
MOVL C00801 V=800.0 PL=0
MOVL C00802 V=800.0 PL=0
MOVL C00803 V=800.0 PL=0
MOVL C00804 V=800.0 PL=0
MOVL C00805 V=800.0 PL=0
MOVL C00806 V=800.0 PL=0
MOVL C00807 V=800.0 PL=0
MOVL C00808 V=800.0 PL=0
MOVL C00809 V=800.0 PL=0
MOVL C00810 V=800.0 PL=0
MOVL C00811 V=800.0 PL=0
MOVL C00812 V=800.0 PL=0
MOVL C00813 V=800.0 PL=0
MOVL C00814 V=800.0 PL=0
MOVL C00815 V=800.0 PL=0
MOVL C00816 V=800.0 PL=0
MOVL C00817 V=800.0 PL=0
MOVL C00818 V=800.0 PL=0
MOVL C00819 V=800.0 PL=0
MOVL C00820 V=800.0 PL=0
MOVL C00821 V=800.0 PL=0
MOVL C00822 V=800.0 PL=0
MOVL C00823 V=800.0 PL=0
MOVL C00824 V=800.0 PL=0
MOVL C00825 V=800.0 PL=0
MOVL C00826 V=800.0 PL=0
MOVL C00827 V=800.0 PL=0
MOVL C00828 V=800.0 PL=0
MOVL C00829 V=800.0 PL=0
MOVL C00830 V=800.0 PL=0
MOVL C00831 V=800.0 PL=0
MOVL C00832 V=800.0 PL=0
MOVL C00833 V=800.0 PL=0
MOVL C00834 V=800.0 PL=0
MOVL C00835 V=800.0 PL=0
MOVL C00836 V=800.0 PL=0
MOVL C00837 V=800.0 PL=0
MOVL C00838 V=800.0 PL=0
MOVL C00839 V=800.0 PL=0
MOVL C00840 V=800.0 PL=0
MOVL C00841 V=800.0 PL=0
MOVL C00842 V=800.0 PL=0
MOVL C00843 V=800.0 PL=0
MOVL C00844 V=800.0 PL=0
MOVL C00845 V=800.0 PL=0
MOVL C00846 V=800.0 PL=0
MOVL C00847 V=800.0 PL=0
MOVL C00848 V=800.0 PL=0
MOVL C00849 V=800.0 PL=0
MOVL C00850 V=800.0 PL=0
MOVL C00851 V=800.0 PL=0
MOVL C00852 V=800.0 PL=0
MOVL C00853 V=800.0 PL=0
MOVL C00854 V=800.0 PL=0
MOVL C00855 V=800.0 PL=0
MOVL C00856 V=800.0 PL=0
MOVL C00857 V=800.0 PL=0
MOVL C00858 V=800.0 PL=0
MOVL C00859 V=800.0 PL=0
MOVL C00860 V=800.0 PL=0
MOVL C00861 V=800.0 PL=0
MOVL C00862 V=800.0 PL=0
MOVL C00863 V=800.0 PL=0
MOVL C00864 V=800.0 PL=0
MOVL C00865 V=800.0 PL=0
MOVL C00866 V=800.0 PL=0
MOVL C00867 V=800.0 PL=0
MOVL C00868 V=800.0 PL=0
MOVL C00869 V=800.0 PL=0
MOVL C00870 V=800.0 PL=0
MOVL C00871 V=800.0 PL=0
MOVL C00872 V=800.0 PL=0
MOVL C00873 V=800.0 PL=0
MOVL C00874 V=800.0 PL=0
MOVL C00875 V=800.0 PL=0
MOVL C00876 V=800.0 PL=0
MOVL C00877 V=800.0 PL=0
MOVL C00878 V=800.0 PL=0
MOVL C00879 V=800.0 PL=0
MOVL C00880 V=800.0 PL=0
MOVL C00881 V=800.0 PL=0
MOVL C00882 V=800.0 PL=0
MOVL C00883 V=800.0 PL=0
MOVL C00884 V=800.0 PL=0
MOVL C00885 V=800.0 PL=0
MOVL C00886 V=800.0 PL=0
MOVL C00887 V=800.0 PL=0
MOVL C00888 V=800.0 PL=0
MOVL C00889 V=800.0 PL=0
MOVL C00890 V=800.0 PL=0
MOVL C00891 V=800.0 PL=0
MOVL C00892 V=800.0 PL=0
MOVL C00893 V=800.0 PL=0
MOVL C00894 V=800.0 PL=0
MOVL C00895 V=800.0 PL=0
MOVL C00896 V=800.0 PL=0
MOVL C00897 V=800.0 PL=0
MOVL C00898 V=800.0 PL=0
MOVL C00899 V=800.0 PL=0
MOVL C00900 V=800.0 PL=0
MOVL C00901 V=800.0 PL=0
MOVL C00902 V=800.0 PL=0
MOVL C00903 V=800.0 PL=0
MOVL C00904 V=800.0 PL=0
MOVL C00905 V=800.0 PL=0
MOVL C00906 V=800.0 PL=0
MOVL C00907 V=800.0 PL=0
MOVL C00908 V=800.0 PL=0
MOVL C00909 V=800.0 PL=0
MOVL C00910 V=800.0 PL=0
MOVL C00911 V=800.0 PL=0
MOVL C00912 V=800.0 PL=0
MOVL C00913 V=800.0 PL=0
MOVL C00914 V=800.0 PL=0
MOVL C00915 V=800.0 PL=0
MOVL C00916 V=800.0 PL=0
MOVL C00917 V=800.0 PL=0
MOVL C00918 V=800.0 PL=0
MOVL C00919 V=800.0 PL=0
MOVL C00920 V=800.0 PL=0
MOVL C00921 V=800.0 PL=0
MOVL C00922 V=800.0 PL=0
MOVL C00923 V=800.0 PL=0
MOVL C00924 V=800.0 PL=0
MOVL C00925 V=800.0 PL=0
MOVL C00926 V=800.0 PL=0
MOVL C00927 V=800.0 PL=0
MOVL C00928 V=800.0 PL=0
MOVL C00929 V=800.0 PL=0
MOVL C00930 V=800.0 PL=0
MOVL C00931 V=800.0 PL=0
MOVL C00932 V=800.0 PL=0
MOVL C00933 V=800.0 PL=0
MOVL C00934 V=800.0 PL=0
MOVL C00935 V=800.0 PL=0
MOVL C00936 V=800.0 PL=0
MOVL C00937 V=800.0 PL=0
MOVL C00938 V=800.0 PL=0
MOVL C00939 V=800.0 PL=0
MOVL C00940 V=800.0 PL=0
MOVL C00941 V=800.0 PL=0
MOVL C00942 V=800.0 PL=0
MOVL C00943 V=800.0 PL=0
MOVL C00944 V=800.0 PL=0
MOVL C00945 V=800.0 PL=0
MOVL C00946 V=800.0 PL=0
MOVL C00947 V=800.0 PL=0
MOVL C00948 V=800.0 PL=0
MOVL C00949 V=800.0 PL=0
MOVL C00950 V=800.0 PL=0
MOVL C00951 V=800.0 PL=0
MOVL C00952 V=800.0 PL=0
MOVL C00953 V=800.0 PL=0
MOVL C00954 V=800.0 PL=0
MOVL C00955 V=800.0 PL=0
MOVL C00956 V=800.0 PL=0
MOVL C00957 V=800.0 PL=0
MOVL C00958 V=800.0 PL=0
MOVL C00959 V=800.0 PL=0
MOVL C00960 V=800.0 PL=0
MOVL C00961 V=800.0 PL=0
MOVL C00962 V=800.0 PL=0
MOVL C00963 V=800.0 PL=0
MOVL C00964 V=800.0 PL=0
MOVL C00965 V=800.0 PL=0
MOVL C00966 V=800.0 PL=0
MOVL C00967 V=800.0 PL=0
MOVL C00968 V=800.0 PL=0
MOVL C00969 V=800.0 PL=0
MOVL C00970 V=800.0 PL=0
MOVL C00971 V=800.0 PL=0
MOVL C00972 V=800.0 PL=0
MOVL C00973 V=800.0 PL=0
MOVL C00974 V=800.0 PL=0
MOVL C00975 V=800.0 PL=0
MOVL C00976 V=800.0 PL=0
MOVL C00977 V=800.0 PL=0
MOVL C00978 V=800.0 PL=0
MOVL C00979 V=800.0 PL=0
MOVL C00980 V=800.0 PL=0
MOVL C00981 V=800.0 PL=0
MOVL C00982 V=800.0 PL=0
MOVL C00983 V=800.0 PL=0
MOVL C00984 V=800.0 PL=0
MOVL C00985 V=800.0 PL=0
MOVL C00986 V=800.0 PL=0
MOVL C00987 V=800.0 PL=0
MOVL C00988 V=800.0 PL=0
MOVL C00989 V=800.0 PL=0
MOVL C00990 V=800.0 PL=0
MOVL C00991 V=800.0 PL=0
MOVL C00992 V=800.0 PL=0
MOVL C00993 V=800.0 PL=0
MOVL C00994 V=800.0 PL=0
MOVL C00995 V=800.0 PL=0
MOVL C00996 V=800.0 PL=0
MOVL C00997 V=800.0 PL=0
MOVL C00998 V=800.0 PL=0
MOVL C00999 V=800.0 PL=0
MOVL C01000 V=800.0 PL=0
MOVL C01001 V=800.0 PL=0
MOVL C01002 V=800.0 PL=0
MOVL C01003 V=800.0 PL=0
MOVL C01004 V=800.0 PL=0
MOVL C01005 V=800.0 PL=0
MOVL C01006 V=800.0 PL=0
MOVL C01007 V=800.0 PL=0
MOVL C01008 V=800.0 PL=0
MOVL C01009 V=800.0 PL=0
MOVL C01010 V=800.0 PL=0
MOVL C01011 V=800.0 PL=0
MOVL C01012 V=800.0 PL=0
MOVL C01013 V=800.0 PL=0
MOVL C01014 V=800.0 PL=0
MOVL C01015 V=800.0 PL=0
MOVL C01016 V=800.0 PL=0
MOVL C01017 V=800.0 PL=0
MOVL C01018 V=800.0 PL=0
MOVL C01019 V=800.0 PL=0
MOVL C01020 V=800.0 PL=0
MOVL C01021 V=800.0 PL=0
MOVL C01022 V=800.0 PL=0
MOVL C01023 V=800.0 PL=0
MOVL C01024 V=800.0 PL=0
MOVL C01025 V=800.0 PL=0
MOVL C01026 V=800.0 PL=0
MOVL C01027 V=800.0 PL=0
MOVL C01028 V=800.0 PL=0
MOVL C01029 V=800.0 PL=0
MOVL C01030 V=800.0 PL=0
MOVL C01031 V=800.0 PL=0
MOVL C01032 V=800.0 PL=0
MOVL C01033 V=800.0 PL=0
MOVL C01034 V=800.0 PL=0
MOVL C01035 V=800.0 PL=0
MOVL C01036 V=800.0 PL=0
MOVL C01037 V=800.0 PL=0
MOVL C01038 V=800.0 PL=0
MOVL C01039 V=800.0 PL=0
MOVL C01040 V=800.0 PL=0
MOVL C01041 V=800.0 PL=0
MOVL C01042 V=800.0 PL=0
MOVL C01043 V=800.0 PL=0
MOVL C01044 V=800.0 PL=0
MOVL C01045 V=800.0 PL=0
MOVL C01046 V=800.0 PL=0
MOVL C01047 V=800.0 PL=0
MOVL C01048 V=800.0 PL=0
MOVL C01049 V=800.0 PL=0
MOVL C01050 V=800.0 PL=0
MOVL C01051 V=800.0 PL=0
MOVL C01052 V=800.0 PL=0
MOVL C01053 V=800.0 PL=0
MOVL C01054 V=800.0 PL=0
MOVL C01055 V=800.0 PL=0
MOVL C01056 V=800.0 PL=0
MOVL C01057 V=800.0 PL=0
MOVL C01058 V=800.0 PL=0
MOVL C01059 V=800.0 PL=0
MOVL C01060 V=800.0 PL=0
MOVL C01061 V=800.0 PL=0
MOVL C01062 V=800.0 PL=0
MOVL C01063 V=800.0 PL=0
MOVL C01064 V=800.0 PL=0
MOVL C01065 V=800.0 PL=0
MOVL C01066 V=800.0 PL=0
MOVL C01067 V=800.0 PL=0
MOVL C01068 V=800.0 PL=0
MOVL C01069 V=800.0 PL=0
MOVL C01070 V=800.0 PL=0
MOVL C01071 V=800.0 PL=0
MOVL C01072 V=800.0 PL=0
MOVL C01073 V=800.0 PL=0
MOVL C01074 V=800.0 PL=0
MOVL C01075 V=800.0 PL=0
MOVL C01076 V=800.0 PL=0
MOVL C01077 V=800.0 PL=0
MOVL C01078 V=800.0 PL=0
MOVL C01079 V=800.0 PL=0
MOVL C01080 V=800.0 PL=0
MOVL C01081 V=800.0 PL=0
MOVL C01082 V=800.0 PL=0
MOVL C01083 V=800.0 PL=0
MOVL C01084 V=800.0 PL=0
MOVL C01085 V=800.0 PL=0
MOVL C01086 V=800.0 PL=0
MOVL C01087 V=800.0 PL=0
MOVL C01088 V=800.0 PL=0
MOVL C01089 V=800.0 PL=0
MOVL C01090 V=800.0 PL=0
MOVL C01091 V=800.0 PL=0
MOVL C01092 V=800.0 PL=0
MOVL C01093 V=800.0 PL=0
MOVL C01094 V=800.0 PL=0
MOVL C01095 V=800.0 PL=0
MOVL C01096 V=800.0 PL=0
MOVL C01097 V=800.0 PL=0
MOVL C01098 V=800.0 PL=0
MOVL C01099 V=800.0 PL=0
MOVL C01100 V=800.0 PL=0
MOVL C01101 V=800.0 PL=0
MOVL C01102 V=800.0 PL=0
MOVL C01103 V=800.0 PL=0
MOVL C01104 V=800.0 PL=0
MOVL C01105 V=800.0 PL=0
MOVL C01106 V=800.0 PL=0
MOVL C01107 V=800.0 PL=0
MOVL C01108 V=800.0 PL=0
MOVL C01109 V=800.0 PL=0
MOVL C01110 V=800.0 PL=0
MOVL C01111 V=800.0 PL=0
MOVL C01112 V=800.0 PL=0
MOVL C01113 V=800.0 PL=0
MOVL C01114 V=800.0 PL=0
MOVL C01115 V=800.0 PL=0
MOVL C01116 V=800.0 PL=0
MOVL C01117 V=800.0 PL=0
MOVL C01118 V=800.0 PL=0
MOVL C01119 V=800.0 PL=0
MOVL C01120 V=800.0 PL=0
MOVL C01121 V=800.0 PL=0
MOVL C01122 V=800.0 PL=0
MOVL C01123 V=800.0 PL=0
MOVL C01124 V=800.0 PL=0
MOVL C01125 V=800.0 PL=0
MOVL C01126 V=800.0 PL=0
MOVL C01127 V=800.0 PL=0
MOVL C01128 V=800.0 PL=0
MOVL C01129 V=800.0 PL=0
MOVL C01130 V=800.0 PL=0
MOVL C01131 V=800.0 PL=0
MOVL C01132 V=800.0 PL=0
MOVL C01133 V=800.0 PL=0
MOVL C01134 V=800.0 PL=0
MOVL C01135 V=800.0 PL=0
MOVL C01136 V=800.0 PL=0
MOVL C01137 V=800.0 PL=0
MOVL C01138 V=800.0 PL=0
MOVL C01139 V=800.0 PL=0
MOVL C01140 V=800.0 PL=0
MOVL C01141 V=800.0 PL=0
MOVL C01142 V=800.0 PL=0
MOVL C01143 V=800.0 PL=0
MOVL C01144 V=800.0 PL=0
MOVL C01145 V=800.0 PL=0
MOVL C01146 V=800.0 PL=0
MOVL C01147 V=800.0 PL=0
MOVL C01148 V=800.0 PL=0
MOVL C01149 V=800.0 PL=0
MOVL C01150 V=800.0 PL=0
MOVL C01151 V=800.0 PL=0
MOVL C01152 V=800.0 PL=0
MOVL C01153 V=800.0 PL=0
MOVL C01154 V=800.0 PL=0
MOVL C01155 V=800.0 PL=0
MOVL C01156 V=800.0 PL=0
MOVL C01157 V=800.0 PL=0
MOVL C01158 V=800.0 PL=0
MOVL C01159 V=800.0 PL=0
MOVL C01160 V=800.0 PL=0
MOVL C01161 V=800.0 PL=0
MOVL C01162 V=800.0 PL=0
MOVL C01163 V=800.0 PL=0
MOVL C01164 V=800.0 PL=0
MOVL C01165 V=800.0 PL=0
MOVL C01166 V=800.0 PL=0
MOVL C01167 V=800.0 PL=0
MOVL C01168 V=800.0 PL=0
MOVL C01169 V=800.0 PL=0
MOVL C01170 V=800.0 PL=0
MOVL C01171 V=800.0 PL=0
MOVL C01172 V=800.0 PL=0
MOVL C01173 V=800.0 PL=0
MOVL C01174 V=800.0 PL=0
MOVL C01175 V=800.0 PL=0
MOVL C01176 V=800.0 PL=0
MOVL C01177 V=800.0 PL=0
MOVL C01178 V=800.0 PL=0
MOVL C01179 V=800.0 PL=0
MOVL C01180 V=800.0 PL=0
MOVL C01181 V=800.0 PL=0
MOVL C01182 V=800.0 PL=0
MOVL C01183 V=800.0 PL=0
MOVL C01184 V=800.0 PL=0
MOVL C01185 V=800.0 PL=0
MOVL C01186 V=800.0 PL=0
MOVL C01187 V=800.0 PL=0
MOVL C01188 V=800.0 PL=0
MOVL C01189 V=800.0 PL=0
MOVL C01190 V=800.0 PL=0
MOVL C01191 V=800.0 PL=0
MOVL C01192 V=800.0 PL=0
MOVL C01193 V=800.0 PL=0
MOVL C01194 V=800.0 PL=0
MOVL C01195 V=800.0 PL=0
MOVL C01196 V=800.0 PL=0
MOVL C01197 V=800.0 PL=0
MOVL C01198 V=800.0 PL=0
MOVL C01199 V=800.0 PL=0
MOVL C01200 V=800.0 PL=0
MOVL C01201 V=800.0 PL=0
MOVL C01202 V=800.0 PL=0
MOVL C01203 V=800.0 PL=0
MOVL C01204 V=800.0 PL=0
MOVL C01205 V=800.0 PL=0
MOVL C01206 V=800.0 PL=0
MOVL C01207 V=800.0 PL=0
MOVL C01208 V=800.0 PL=0
MOVL C01209 V=800.0 PL=0
MOVL C01210 V=800.0 PL=0
MOVL C01211 V=800.0 PL=0
MOVL C01212 V=800.0 PL=0
MOVL C01213 V=800.0 PL=0
MOVL C01214 V=800.0 PL=0
MOVL C01215 V=800.0 PL=0
MOVL C01216 V=800.0 PL=0
MOVL C01217 V=800.0 PL=0
MOVL C01218 V=800.0 PL=0
MOVL C01219 V=800.0 PL=0
MOVL C01220 V=800.0 PL=0
MOVL C01221 V=800.0 PL=0
MOVL C01222 V=800.0 PL=0
MOVL C01223 V=800.0 PL=0
MOVL C01224 V=800.0 PL=0
MOVL C01225 V=800.0 PL=0
MOVL C01226 V=800.0 PL=0
MOVL C01227 V=800.0 PL=0
MOVL C01228 V=800.0 PL=0
MOVL C01229 V=800.0 PL=0
MOVL C01230 V=800.0 PL=0
MOVL C01231 V=800.0 PL=0
MOVL C01232 V=800.0 PL=0
MOVL C01233 V=800.0 PL=0
MOVL C01234 V=800.0 PL=0
MOVL C01235 V=800.0 PL=0
MOVL C01236 V=800.0 PL=0
MOVL C01237 V=800.0 PL=0
MOVL C01238 V=800.0 PL=0
MOVL C01239 V=800.0 PL=0
MOVL C01240 V=800.0 PL=0
MOVL C01241 V=800.0 PL=0
MOVL C01242 V=800.0 PL=0
MOVL C01243 V=800.0 PL=0
MOVL C01244 V=800.0 PL=0
MOVL C01245 V=800.0 PL=0
MOVL C01246 V=800.0 PL=0
MOVL C01247 V=800.0 PL=0
MOVL C01248 V=800.0 PL=0
MOVL C01249 V=800.0 PL=0
MOVL C01250 V=800.0 PL=0
MOVL C01251 V=800.0 PL=0
MOVL C01252 V=800.0 PL=0
MOVL C01253 V=800.0 PL=0
MOVL C01254 V=800.0 PL=0
MOVL C01255 V=800.0 PL=0
MOVL C01256 V=800.0 PL=0
MOVL C01257 V=800.0 PL=0
MOVL C01258 V=800.0 PL=0
MOVL C01259 V=800.0 PL=0
MOVL C01260 V=800.0 PL=0
MOVL C01261 V=800.0 PL=0
MOVL C01262 V=800.0 PL=0
MOVL C01263 V=800.0 PL=0
MOVL C01264 V=800.0 PL=0
MOVL C01265 V=800.0 PL=0
MOVL C01266 V=800.0 PL=0
MOVL C01267 V=800.0 PL=0
MOVL C01268 V=800.0 PL=0
MOVL C01269 V=800.0 PL=0
MOVL C01270 V=800.0 PL=0
MOVL C01271 V=800.0 PL=0
MOVL C01272 V=800.0 PL=0
MOVL C01273 V=800.0 PL=0
MOVL C01274 V=800.0 PL=0
MOVL C01275 V=800.0 PL=0
MOVL C01276 V=800.0 PL=0
MOVL C01277 V=800.0 PL=0
MOVL C01278 V=800.0 PL=0
MOVL C01279 V=800.0 PL=0
MOVL C01280 V=800.0 PL=0
MOVL C01281 V=800.0 PL=0
MOVL C01282 V=800.0 PL=0
MOVL C01283 V=800.0 PL=0
MOVL C01284 V=800.0 PL=0
MOVL C01285 V=800.0 PL=0
MOVL C01286 V=800.0 PL=0
MOVL C01287 V=800.0 PL=0
MOVL C01288 V=800.0 PL=0
MOVL C01289 V=800.0 PL=0
MOVL C01290 V=800.0 PL=0
MOVL C01291 V=800.0 PL=0
MOVL C01292 V=800.0 PL=0
MOVL C01293 V=800.0 PL=0
MOVL C01294 V=800.0 PL=0
MOVL C01295 V=800.0 PL=0
MOVL C01296 V=800.0 PL=0
MOVL C01297 V=800.0 PL=0
MOVL C01298 V=800.0 PL=0
MOVL C01299 V=800.0 PL=0
MOVL C01300 V=800.0 PL=0
MOVL C01301 V=800.0 PL=0
MOVL C01302 V=800.0 PL=0
MOVL C01303 V=800.0 PL=0
MOVL C01304 V=800.0 PL=0
MOVL C01305 V=800.0 PL=0
MOVL C01306 V=800.0 PL=0
MOVL C01307 V=800.0 PL=0
MOVL C01308 V=800.0 PL=0
MOVL C01309 V=800.0 PL=0
MOVL C01310 V=800.0 PL=0
MOVL C01311 V=800.0 PL=0
MOVL C01312 V=800.0 PL=0
MOVL C01313 V=800.0 PL=0
MOVL C01314 V=800.0 PL=0
MOVL C01315 V=800.0 PL=0
MOVL C01316 V=800.0 PL=0
MOVL C01317 V=800.0 PL=0
MOVL C01318 V=800.0 PL=0
MOVL C01319 V=800.0 PL=0
MOVL C01320 V=800.0 PL=0
MOVL C01321 V=800.0 PL=0
MOVL C01322 V=800.0 PL=0
MOVL C01323 V=800.0 PL=0
MOVL C01324 V=800.0 PL=0
MOVL C01325 V=800.0 PL=0
MOVL C01326 V=800.0 PL=0
MOVL C01327 V=800.0 PL=0
MOVL C01328 V=800.0 PL=0
MOVL C01329 V=800.0 PL=0
MOVL C01330 V=800.0 PL=0
MOVL C01331 V=800.0 PL=0
MOVL C01332 V=800.0 PL=0
MOVL C01333 V=800.0 PL=0
MOVL C01334 V=800.0 PL=0
MOVL C01335 V=800.0 PL=0
MOVL C01336 V=800.0 PL=0
MOVL C01337 V=800.0 PL=0
MOVL C01338 V=800.0 PL=0
MOVL C01339 V=800.0 PL=0
MOVL C01340 V=800.0 PL=0
MOVL C01341 V=800.0 PL=0
MOVL C01342 V=800.0 PL=0
MOVL C01343 V=800.0 PL=0
MOVL C01344 V=800.0 PL=0
MOVL C01345 V=800.0 PL=0
MOVL C01346 V=800.0 PL=0
MOVL C01347 V=800.0 PL=0
MOVL C01348 V=800.0 PL=0
MOVL C01349 V=800.0 PL=0
MOVL C01350 V=800.0 PL=0
MOVL C01351 V=800.0 PL=0
MOVL C01352 V=800.0 PL=0
MOVL C01353 V=800.0 PL=0
MOVL C01354 V=800.0 PL=0
MOVL C01355 V=800.0 PL=0
MOVL C01356 V=800.0 PL=0
MOVL C01357 V=800.0 PL=0
MOVL C01358 V=800.0 PL=0
MOVL C01359 V=800.0 PL=0
MOVL C01360 V=800.0 PL=0
MOVL C01361 V=800.0 PL=0
MOVL C01362 V=800.0 PL=0
MOVL C01363 V=800.0 PL=0
MOVL C01364 V=800.0 PL=0
MOVL C01365 V=800.0 PL=0
MOVL C01366 V=800.0 PL=0
MOVL C01367 V=800.0 PL=0
MOVL C01368 V=800.0 PL=0
MOVL C01369 V=800.0 PL=0
MOVL C01370 V=800.0 PL=0
MOVL C01371 V=800.0 PL=0
MOVL C01372 V=800.0 PL=0
MOVL C01373 V=800.0 PL=0
MOVL C01374 V=800.0 PL=0
MOVL C01375 V=800.0 PL=0
MOVL C01376 V=800.0 PL=0
MOVL C01377 V=800.0 PL=0
MOVL C01378 V=800.0 PL=0
MOVL C01379 V=800.0 PL=0
MOVL C01380 V=800.0 PL=0
MOVL C01381 V=800.0 PL=0
MOVL C01382 V=800.0 PL=0
MOVL C01383 V=800.0 PL=0
MOVL C01384 V=800.0 PL=0
MOVL C01385 V=800.0 PL=0
MOVL C01386 V=800.0 PL=0
MOVL C01387 V=800.0 PL=0
MOVL C01388 V=800.0 PL=0
MOVL C01389 V=800.0 PL=0
MOVL C01390 V=800.0 PL=0
MOVL C01391 V=800.0 PL=0
MOVL C01392 V=800.0 PL=0
MOVL C01393 V=800.0 PL=0
MOVL C01394 V=800.0 PL=0
MOVL C01395 V=800.0 PL=0
MOVL C01396 V=800.0 PL=0
MOVL C01397 V=800.0 PL=0
MOVL C01398 V=800.0 PL=0
MOVL C01399 V=800.0 PL=0
MOVL C01400 V=800.0 PL=0
MOVL C01401 V=800.0 PL=0
MOVL C01402 V=800.0 PL=0
MOVL C01403 V=800.0 PL=0
MOVL C01404 V=800.0 PL=0
MOVL C01405 V=800.0 PL=0
MOVL C01406 V=800.0 PL=0
MOVL C01407 V=800.0 PL=0
MOVL C01408 V=800.0 PL=0
MOVL C01409 V=800.0 PL=0
MOVL C01410 V=800.0 PL=0
MOVL C01411 V=800.0 PL=0
MOVL C01412 V=800.0 PL=0
MOVL C01413 V=800.0 PL=0
MOVL C01414 V=800.0 PL=0
MOVL C01415 V=800.0 PL=0
MOVL C01416 V=800.0 PL=0
MOVL C01417 V=800.0 PL=0
MOVL C01418 V=800.0 PL=0
MOVL C01419 V=800.0 PL=0
MOVL C01420 V=800.0 PL=0
MOVL C01421 V=800.0 PL=0
MOVL C01422 V=800.0 PL=0
MOVL C01423 V=800.0 PL=0
MOVL C01424 V=800.0 PL=0
MOVL C01425 V=800.0 PL=0
MOVL C01426 V=800.0 PL=0
MOVL C01427 V=800.0 PL=0
MOVL C01428 V=800.0 PL=0
MOVL C01429 V=800.0 PL=0
MOVL C01430 V=800.0 PL=0
MOVL C01431 V=800.0 PL=0
MOVL C01432 V=800.0 PL=0
MOVL C01433 V=800.0 PL=0
MOVL C01434 V=800.0 PL=0
MOVL C01435 V=800.0 PL=0
MOVL C01436 V=800.0 PL=0
MOVL C01437 V=800.0 PL=0
MOVL C01438 V=800.0 PL=0
MOVL C01439 V=800.0 PL=0
MOVL C01440 V=800.0 PL=0
MOVL C01441 V=800.0 PL=0
MOVL C01442 V=800.0 PL=0
MOVL C01443 V=800.0 PL=0
MOVL C01444 V=800.0 PL=0
MOVL C01445 V=800.0 PL=0
MOVL C01446 V=800.0 PL=0
MOVL C01447 V=800.0 PL=0
MOVL C01448 V=800.0 PL=0
MOVL C01449 V=800.0 PL=0
MOVL C01450 V=800.0 PL=0
MOVL C01451 V=800.0 PL=0
MOVL C01452 V=800.0 PL=0
MOVL C01453 V=800.0 PL=0
MOVL C01454 V=800.0 PL=0
MOVL C01455 V=800.0 PL=0
MOVL C01456 V=800.0 PL=0
MOVL C01457 V=800.0 PL=0
MOVL C01458 V=800.0 PL=0
MOVL C01459 V=800.0 PL=0
MOVL C01460 V=800.0 PL=0
MOVL C01461 V=800.0 PL=0
MOVL C01462 V=800.0 PL=0
MOVL C01463 V=800.0 PL=0
MOVL C01464 V=800.0 PL=0
MOVL C01465 V=800.0 PL=0
MOVL C01466 V=800.0 PL=0
MOVL C01467 V=800.0 PL=0
MOVL C01468 V=800.0 PL=0
MOVL C01469 V=800.0 PL=0
MOVL C01470 V=800.0 PL=0
MOVL C01471 V=800.0 PL=0
MOVL C01472 V=800.0 PL=0
MOVL C01473 V=800.0 PL=0
MOVL C01474 V=800.0 PL=0
MOVL C01475 V=800.0 PL=0
MOVL C01476 V=800.0 PL=0
MOVL C01477 V=800.0 PL=0
MOVL C01478 V=800.0 PL=0
MOVL C01479 V=800.0 PL=0
MOVL C01480 V=800.0 PL=0
MOVL C01481 V=800.0 PL=0
MOVL C01482 V=800.0 PL=0
MOVL C01483 V=800.0 PL=0
MOVL C01484 V=800.0 PL=0
MOVL C01485 V=800.0 PL=0
MOVL C01486 V=800.0 PL=0
MOVL C01487 V=800.0 PL=0
MOVL C01488 V=800.0 PL=0
MOVL C01489 V=800.0 PL=0
MOVL C01490 V=800.0 PL=0
MOVL C01491 V=800.0 PL=0
MOVL C01492 V=800.0 PL=0
MOVL C01493 V=800.0 PL=0
MOVL C01494 V=800.0 PL=0
MOVL C01495 V=800.0 PL=0
MOVL C01496 V=800.0 PL=0
MOVL C01497 V=800.0 PL=0
MOVL C01498 V=800.0 PL=0
MOVL C01499 V=800.0 PL=0
MOVL C01500 V=800.0 PL=0
MOVL C01501 V=800.0 PL=0
MOVL C01502 V=800.0 PL=0
MOVL C01503 V=800.0 PL=0
MOVL C01504 V=800.0 PL=0
MOVL C01505 V=800.0 PL=0
MOVL C01506 V=800.0 PL=0
MOVL C01507 V=800.0 PL=0
MOVL C01508 V=800.0 PL=0
MOVL C01509 V=800.0 PL=0
MOVL C01510 V=800.0 PL=0
MOVL C01511 V=800.0 PL=0
MOVL C01512 V=800.0 PL=0
MOVL C01513 V=800.0 PL=0
MOVL C01514 V=800.0 PL=0
MOVL C01515 V=800.0 PL=0
MOVL C01516 V=800.0 PL=0
MOVL C01517 V=800.0 PL=0
MOVL C01518 V=800.0 PL=0
MOVL C01519 V=800.0 PL=0
MOVL C01520 V=800.0 PL=0
MOVL C01521 V=800.0 PL=0
MOVL C01522 V=800.0 PL=0
MOVL C01523 V=800.0 PL=0
MOVL C01524 V=800.0 PL=0
MOVL C01525 V=800.0 PL=0
MOVL C01526 V=800.0 PL=0
MOVL C01527 V=800.0 PL=0
MOVL C01528 V=800.0 PL=0
MOVL C01529 V=800.0 PL=0
MOVL C01530 V=800.0 PL=0
MOVL C01531 V=800.0 PL=0
MOVL C01532 V=800.0 PL=0
MOVL C01533 V=800.0 PL=0
MOVL C01534 V=800.0 PL=0
MOVL C01535 V=800.0 PL=0
MOVL C01536 V=800.0 PL=0
MOVL C01537 V=800.0 PL=0
MOVL C01538 V=800.0 PL=0
MOVL C01539 V=800.0 PL=0
MOVL C01540 V=800.0 PL=0
MOVL C01541 V=800.0 PL=0
MOVL C01542 V=800.0 PL=0
MOVL C01543 V=800.0 PL=0
MOVL C01544 V=800.0 PL=0
MOVL C01545 V=800.0 PL=0
MOVL C01546 V=800.0 PL=0
MOVL C01547 V=800.0 PL=0
MOVL C01548 V=800.0 PL=0
MOVL C01549 V=800.0 PL=0
MOVL C01550 V=800.0 PL=0
MOVL C01551 V=800.0 PL=0
MOVL C01552 V=800.0 PL=0
MOVL C01553 V=800.0 PL=0
MOVL C01554 V=800.0 PL=0
MOVL C01555 V=800.0 PL=0
MOVL C01556 V=800.0 PL=0
MOVL C01557 V=800.0 PL=0
MOVL C01558 V=800.0 PL=0
MOVL C01559 V=800.0 PL=0
MOVL C01560 V=800.0 PL=0
MOVL C01561 V=800.0 PL=0
MOVL C01562 V=800.0 PL=0
MOVL C01563 V=800.0 PL=0
MOVL C01564 V=800.0 PL=0
MOVL C01565 V=800.0 PL=0
MOVL C01566 V=800.0 PL=0
MOVL C01567 V=800.0 PL=0
MOVL C01568 V=800.0 PL=0
MOVL C01569 V=800.0 PL=0
MOVL C01570 V=800.0 PL=0
MOVL C01571 V=800.0 PL=0
MOVL C01572 V=800.0 PL=0
MOVL C01573 V=800.0 PL=0
MOVL C01574 V=800.0 PL=0
MOVL C01575 V=800.0 PL=0
MOVL C01576 V=800.0 PL=0
MOVL C01577 V=800.0 PL=0
MOVL C01578 V=800.0 PL=0
MOVL C01579 V=800.0 PL=0
MOVL C01580 V=800.0 PL=0
MOVL C01581 V=800.0 PL=0
MOVL C01582 V=800.0 PL=0
MOVL C01583 V=800.0 PL=0
MOVL C01584 V=800.0 PL=0
MOVL C01585 V=800.0 PL=0
MOVL C01586 V=800.0 PL=0
MOVL C01587 V=800.0 PL=0
MOVL C01588 V=800.0 PL=0
MOVL C01589 V=800.0 PL=0
MOVL C01590 V=800.0 PL=0
MOVL C01591 V=800.0 PL=0
MOVL C01592 V=800.0 PL=0
MOVL C01593 V=800.0 PL=0
MOVL C01594 V=800.0 PL=0
MOVL C01595 V=800.0 PL=0
MOVL C01596 V=800.0 PL=0
MOVL C01597 V=800.0 PL=0
MOVL C01598 V=800.0 PL=0
MOVL C01599 V=800.0 PL=0
MOVL C01600 V=800.0 PL=0
MOVL C01601 V=800.0 PL=0
MOVL C01602 V=800.0 PL=0
MOVL C01603 V=800.0 PL=0
MOVL C01604 V=800.0 PL=0
MOVL C01605 V=800.0 PL=0
MOVL C01606 V=800.0 PL=0
MOVL C01607 V=800.0 PL=0
MOVL C01608 V=800.0 PL=0
MOVL C01609 V=800.0 PL=0
MOVL C01610 V=800.0 PL=0
MOVL C01611 V=800.0 PL=0
MOVL C01612 V=800.0 PL=0
MOVL C01613 V=800.0 PL=0
MOVL C01614 V=800.0 PL=0
MOVL C01615 V=800.0 PL=0
MOVL C01616 V=800.0 PL=0
MOVL C01617 V=800.0 PL=0
MOVL C01618 V=800.0 PL=0
MOVL C01619 V=800.0 PL=0
MOVL C01620 V=800.0 PL=0
MOVL C01621 V=800.0 PL=0
MOVL C01622 V=800.0 PL=0
MOVL C01623 V=800.0 PL=0
MOVL C01624 V=800.0 PL=0
MOVL C01625 V=800.0 PL=0
MOVL C01626 V=800.0 PL=0
MOVL C01627 V=800.0 PL=0
MOVL C01628 V=800.0 PL=0
MOVL C01629 V=800.0 PL=0
MOVL C01630 V=800.0 PL=0
MOVL C01631 V=800.0 PL=0
MOVL C01632 V=800.0 PL=0
MOVL C01633 V=800.0 PL=0
MOVL C01634 V=800.0 PL=0
MOVL C01635 V=800.0 PL=0
MOVL C01636 V=800.0 PL=0
MOVL C01637 V=800.0 PL=0
MOVL C01638 V=800.0 PL=0
MOVL C01639 V=800.0 PL=0
MOVL C01640 V=800.0 PL=0
MOVL C01641 V=800.0 PL=0
MOVL C01642 V=800.0 PL=0
MOVL C01643 V=800.0 PL=0
MOVL C01644 V=800.0 PL=0
MOVL C01645 V=800.0 PL=0
MOVL C01646 V=800.0 PL=0
MOVL C01647 V=800.0 PL=0
MOVL C01648 V=800.0 PL=0
MOVL C01649 V=800.0 PL=0
MOVL C01650 V=800.0 PL=0
MOVL C01651 V=800.0 PL=0
MOVL C01652 V=800.0 PL=0
MOVL C01653 V=800.0 PL=0
MOVL C01654 V=800.0 PL=0
MOVL C01655 V=800.0 PL=0
MOVL C01656 V=800.0 PL=0
MOVL C01657 V=800.0 PL=0
MOVL C01658 V=800.0 PL=0
MOVL C01659 V=800.0 PL=0
MOVL C01660 V=800.0 PL=0
MOVL C01661 V=800.0 PL=0
MOVL C01662 V=800.0 PL=0
MOVL C01663 V=800.0 PL=0
MOVL C01664 V=800.0 PL=0
MOVL C01665 V=800.0 PL=0
MOVL C01666 V=800.0 PL=0
MOVL C01667 V=800.0 PL=0
MOVL C01668 V=800.0 PL=0
MOVL C01669 V=800.0 PL=0
MOVL C01670 V=800.0 PL=0
MOVL C01671 V=800.0 PL=0
MOVL C01672 V=800.0 PL=0
MOVL C01673 V=800.0 PL=0
MOVL C01674 V=800.0 PL=0
MOVL C01675 V=800.0 PL=0
MOVL C01676 V=800.0 PL=0
MOVL C01677 V=800.0 PL=0
MOVL C01678 V=800.0 PL=0
MOVL C01679 V=800.0 PL=0
MOVL C01680 V=800.0 PL=0
MOVL C01681 V=800.0 PL=0
MOVL C01682 V=800.0 PL=0
MOVL C01683 V=800.0 PL=0
MOVL C01684 V=800.0 PL=0
MOVL C01685 V=800.0 PL=0
MOVL C01686 V=800.0 PL=0
MOVL C01687 V=800.0 PL=0
MOVL C01688 V=800.0 PL=0
MOVL C01689 V=800.0 PL=0
MOVL C01690 V=800.0 PL=0
MOVL C01691 V=800.0 PL=0
MOVL C01692 V=800.0 PL=0
MOVL C01693 V=800.0 PL=0
MOVL C01694 V=800.0 PL=0
MOVL C01695 V=800.0 PL=0
MOVL C01696 V=800.0 PL=0
MOVL C01697 V=800.0 PL=0
MOVL C01698 V=800.0 PL=0
MOVL C01699 V=800.0 PL=0
MOVL C01700 V=800.0 PL=0
MOVL C01701 V=800.0 PL=0
MOVL C01702 V=800.0 PL=0
MOVL C01703 V=800.0 PL=0
MOVL C01704 V=800.0 PL=0
MOVL C01705 V=800.0 PL=0
MOVL C01706 V=800.0 PL=0
MOVL C01707 V=800.0 PL=0
MOVL C01708 V=800.0 PL=0
MOVL C01709 V=800.0 PL=0
MOVL C01710 V=800.0 PL=0
MOVL C01711 V=800.0 PL=0
MOVL C01712 V=800.0 PL=0
MOVL C01713 V=800.0 PL=0
MOVL C01714 V=800.0 PL=0
MOVL C01715 V=800.0 PL=0
MOVL C01716 V=800.0 PL=0
MOVL C01717 V=800.0 PL=0
MOVL C01718 V=800.0 PL=0
MOVL C01719 V=800.0 PL=0
MOVL C01720 V=800.0 PL=0
MOVL C01721 V=800.0 PL=0
MOVL C01722 V=800.0 PL=0
MOVL C01723 V=800.0 PL=0
MOVL C01724 V=800.0 PL=0
MOVL C01725 V=800.0 PL=0
MOVL C01726 V=800.0 PL=0
MOVL C01727 V=800.0 PL=0
MOVL C01728 V=800.0 PL=0
MOVL C01729 V=800.0 PL=0
MOVL C01730 V=800.0 PL=0
MOVL C01731 V=800.0 PL=0
MOVL C01732 V=800.0 PL=0
MOVL C01733 V=800.0 PL=0
MOVL C01734 V=800.0 PL=0
MOVL C01735 V=800.0 PL=0
MOVL C01736 V=800.0 PL=0
MOVL C01737 V=800.0 PL=0
MOVL C01738 V=800.0 PL=0
MOVL C01739 V=800.0 PL=0
MOVL C01740 V=800.0 PL=0
MOVL C01741 V=800.0 PL=0
MOVL C01742 V=800.0 PL=0
MOVL C01743 V=800.0 PL=0
MOVL C01744 V=800.0 PL=0
MOVL C01745 V=800.0 PL=0
MOVL C01746 V=800.0 PL=0
MOVL C01747 V=800.0 PL=0
MOVL C01748 V=800.0 PL=0
MOVL C01749 V=800.0 PL=0
MOVL C01750 V=800.0 PL=0
MOVL C01751 V=800.0 PL=0
MOVL C01752 V=800.0 PL=0
MOVL C01753 V=800.0 PL=0
MOVL C01754 V=800.0 PL=0
MOVL C01755 V=800.0 PL=0
MOVL C01756 V=800.0 PL=0
MOVL C01757 V=800.0 PL=0
MOVL C01758 V=800.0 PL=0
MOVL C01759 V=800.0 PL=0
MOVL C01760 V=800.0 PL=0
MOVL C01761 V=800.0 PL=0
MOVL C01762 V=800.0 PL=0
MOVL C01763 V=800.0 PL=0
MOVL C01764 V=800.0 PL=0
MOVL C01765 V=800.0 PL=0
MOVL C01766 V=800.0 PL=0
MOVL C01767 V=800.0 PL=0
MOVL C01768 V=800.0 PL=0
MOVL C01769 V=800.0 PL=0
MOVL C01770 V=800.0 PL=0
MOVL C01771 V=800.0 PL=0
MOVL C01772 V=800.0 PL=0
MOVL C01773 V=800.0 PL=0
MOVL C01774 V=800.0 PL=0
MOVL C01775 V=800.0 PL=0
MOVL C01776 V=800.0 PL=0
MOVL C01777 V=800.0 PL=0
MOVL C01778 V=800.0 PL=0
MOVL C01779 V=800.0 PL=0
MOVL C01780 V=800.0 PL=0
MOVL C01781 V=800.0 PL=0
MOVL C01782 V=800.0 PL=0
MOVL C01783 V=800.0 PL=0
MOVL C01784 V=800.0 PL=0
MOVL C01785 V=800.0 PL=0
MOVL C01786 V=800.0 PL=0
MOVL C01787 V=800.0 PL=0
MOVL C01788 V=800.0 PL=0
MOVL C01789 V=800.0 PL=0
MOVL C01790 V=800.0 PL=0
MOVL C01791 V=800.0 PL=0
MOVL C01792 V=800.0 PL=0
MOVL C01793 V=800.0 PL=0
MOVL C01794 V=800.0 PL=0
MOVL C01795 V=800.0 PL=0
MOVL C01796 V=800.0 PL=0
MOVL C01797 V=800.0 PL=0
MOVL C01798 V=800.0 PL=0
MOVL C01799 V=800.0 PL=0
MOVL C01800 V=800.0 PL=0
MOVL C01801 V=800.0 PL=0
MOVL C01802 V=800.0 PL=0
MOVL C01803 V=800.0 PL=0
MOVL C01804 V=800.0 PL=0
MOVL C01805 V=800.0 PL=0
MOVL C01806 V=800.0 PL=0
MOVL C01807 V=800.0 PL=0
MOVL C01808 V=800.0 PL=0
MOVL C01809 V=800.0 PL=0
MOVL C01810 V=800.0 PL=0
MOVL C01811 V=800.0 PL=0
MOVL C01812 V=800.0 PL=0
MOVL C01813 V=800.0 PL=0
MOVL C01814 V=800.0 PL=0
MOVL C01815 V=800.0 PL=0
MOVL C01816 V=800.0 PL=0
MOVL C01817 V=800.0 PL=0
MOVL C01818 V=800.0 PL=0
MOVL C01819 V=800.0 PL=0
MOVL C01820 V=800.0 PL=0
MOVL C01821 V=800.0 PL=0
MOVL C01822 V=800.0 PL=0
MOVL C01823 V=800.0 PL=0
MOVL C01824 V=800.0 PL=0
MOVL C01825 V=800.0 PL=0
MOVL C01826 V=800.0 PL=0
MOVL C01827 V=800.0 PL=0
MOVL C01828 V=800.0 PL=0
MOVL C01829 V=800.0 PL=0
MOVL C01830 V=800.0 PL=0
MOVL C01831 V=800.0 PL=0
MOVL C01832 V=800.0 PL=0
MOVL C01833 V=800.0 PL=0
MOVL C01834 V=800.0 PL=0
MOVL C01835 V=800.0 PL=0
MOVL C01836 V=800.0 PL=0
MOVL C01837 V=800.0 PL=0
MOVL C01838 V=800.0 PL=0
MOVL C01839 V=800.0 PL=0
MOVL C01840 V=800.0 PL=0
MOVL C01841 V=800.0 PL=0
MOVL C01842 V=800.0 PL=0
MOVL C01843 V=800.0 PL=0
MOVL C01844 V=800.0 PL=0
MOVL C01845 V=800.0 PL=0
MOVL C01846 V=800.0 PL=0
MOVL C01847 V=800.0 PL=0
MOVL C01848 V=800.0 PL=0
MOVL C01849 V=800.0 PL=0
MOVL C01850 V=800.0 PL=0
MOVL C01851 V=800.0 PL=0
MOVL C01852 V=800.0 PL=0
MOVL C01853 V=800.0 PL=0
MOVL C01854 V=800.0 PL=0
MOVL C01855 V=800.0 PL=0
MOVL C01856 V=800.0 PL=0
MOVL C01857 V=800.0 PL=0
MOVL C01858 V=800.0 PL=0
MOVL C01859 V=800.0 PL=0
MOVL C01860 V=800.0 PL=0
MOVL C01861 V=800.0 PL=0
MOVL C01862 V=800.0 PL=0
MOVL C01863 V=800.0 PL=0
MOVL C01864 V=800.0 PL=0
MOVL C01865 V=800.0 PL=0
MOVL C01866 V=800.0 PL=0
MOVL C01867 V=800.0 PL=0
MOVL C01868 V=800.0 PL=0
MOVL C01869 V=800.0 PL=0
MOVL C01870 V=800.0 PL=0
MOVL C01871 V=800.0 PL=0
MOVL C01872 V=800.0 PL=0
MOVL C01873 V=800.0 PL=0
MOVL C01874 V=800.0 PL=0
MOVL C01875 V=800.0 PL=0
MOVL C01876 V=800.0 PL=0
MOVL C01877 V=800.0 PL=0
MOVL C01878 V=800.0 PL=0
MOVL C01879 V=800.0 PL=0
MOVL C01880 V=800.0 PL=0
MOVL C01881 V=800.0 PL=0
MOVL C01882 V=800.0 PL=0
MOVL C01883 V=800.0 PL=0
MOVL C01884 V=800.0 PL=0
MOVL C01885 V=800.0 PL=0
MOVL C01886 V=800.0 PL=0
MOVL C01887 V=800.0 PL=0
MOVL C01888 V=800.0 PL=0
MOVL C01889 V=800.0 PL=0
MOVL C01890 V=800.0 PL=0
MOVL C01891 V=800.0 PL=0
MOVL C01892 V=800.0 PL=0
MOVL C01893 V=800.0 PL=0
MOVL C01894 V=800.0 PL=0
MOVL C01895 V=800.0 PL=0
MOVL C01896 V=800.0 PL=0
MOVL C01897 V=800.0 PL=0
MOVL C01898 V=800.0 PL=0
MOVL C01899 V=800.0 PL=0
MOVL C01900 V=800.0 PL=0
MOVL C01901 V=800.0 PL=0
MOVL C01902 V=800.0 PL=0
MOVL C01903 V=800.0 PL=0
MOVL C01904 V=800.0 PL=0
MOVL C01905 V=800.0 PL=0
MOVL C01906 V=800.0 PL=0
MOVL C01907 V=800.0 PL=0
MOVL C01908 V=800.0 PL=0
MOVL C01909 V=800.0 PL=0
MOVL C01910 V=800.0 PL=0
MOVL C01911 V=800.0 PL=0
MOVL C01912 V=800.0 PL=0
MOVL C01913 V=800.0 PL=0
MOVL C01914 V=800.0 PL=0
MOVL C01915 V=800.0 PL=0
MOVL C01916 V=800.0 PL=0
MOVL C01917 V=800.0 PL=0
MOVL C01918 V=800.0 PL=0
MOVL C01919 V=800.0 PL=0
MOVL C01920 V=800.0 PL=0
MOVL C01921 V=800.0 PL=0
MOVL C01922 V=800.0 PL=0
MOVL C01923 V=800.0 PL=0
MOVL C01924 V=800.0 PL=0
MOVL C01925 V=800.0 PL=0
MOVL C01926 V=800.0 PL=0
MOVL C01927 V=800.0 PL=0
MOVL C01928 V=800.0 PL=0
MOVL C01929 V=800.0 PL=0
MOVL C01930 V=800.0 PL=0
MOVL C01931 V=800.0 PL=0
MOVL C01932 V=800.0 PL=0
MOVL C01933 V=800.0 PL=0
MOVL C01934 V=800.0 PL=0
MOVL C01935 V=800.0 PL=0
MOVL C01936 V=800.0 PL=0
MOVL C01937 V=800.0 PL=0
MOVL C01938 V=800.0 PL=0
MOVL C01939 V=800.0 PL=0
MOVL C01940 V=800.0 PL=0
MOVL C01941 V=800.0 PL=0
MOVL C01942 V=800.0 PL=0
MOVL C01943 V=800.0 PL=0
MOVL C01944 V=800.0 PL=0
MOVL C01945 V=800.0 PL=0
MOVL C01946 V=800.0 PL=0
MOVL C01947 V=800.0 PL=0
MOVL C01948 V=800.0 PL=0
MOVL C01949 V=800.0 PL=0
MOVL C01950 V=800.0 PL=0
MOVL C01951 V=800.0 PL=0
MOVL C01952 V=800.0 PL=0
MOVL C01953 V=800.0 PL=0
MOVL C01954 V=800.0 PL=0
MOVL C01955 V=800.0 PL=0
MOVL C01956 V=800.0 PL=0
MOVL C01957 V=800.0 PL=0
MOVL C01958 V=800.0 PL=0
MOVL C01959 V=800.0 PL=0
MOVL C01960 V=800.0 PL=0
MOVL C01961 V=800.0 PL=0
MOVL C01962 V=800.0 PL=0
MOVL C01963 V=800.0 PL=0
MOVL C01964 V=800.0 PL=0
MOVL C01965 V=800.0 PL=0
MOVL C01966 V=800.0 PL=0
MOVL C01967 V=800.0 PL=0
MOVL C01968 V=800.0 PL=0
MOVL C01969 V=800.0 PL=0
MOVL C01970 V=800.0 PL=0
MOVL C01971 V=800.0 PL=0
MOVL C01972 V=800.0 PL=0
MOVL C01973 V=800.0 PL=0
MOVL C01974 V=800.0 PL=0
MOVL C01975 V=800.0 PL=0
MOVL C01976 V=800.0 PL=0
MOVL C01977 V=800.0 PL=0
MOVL C01978 V=800.0 PL=0
MOVL C01979 V=800.0 PL=0
MOVL C01980 V=800.0 PL=0
MOVL C01981 V=800.0 PL=0
MOVL C01982 V=800.0 PL=0
MOVL C01983 V=800.0 PL=0
MOVL C01984 V=800.0 PL=0
MOVL C01985 V=800.0 PL=0
MOVL C01986 V=800.0 PL=0
MOVL C01987 V=800.0 PL=0
MOVL C01988 V=800.0 PL=0
MOVL C01989 V=800.0 PL=0
MOVL C01990 V=800.0 PL=0
MOVL C01991 V=800.0 PL=0
MOVL C01992 V=800.0 PL=0
MOVL C01993 V=800.0 PL=0
MOVL C01994 V=800.0 PL=0
MOVL C01995 V=800.0 PL=0
MOVL C01996 V=800.0 PL=0
MOVL C01997 V=800.0 PL=0
MOVL C01998 V=800.0 PL=0
MOVL C01999 V=800.0 PL=0
MOVL C02000 V=800.0 PL=0
MOVL C02001 V=800.0 PL=0
MOVL C02002 V=800.0 PL=0
MOVL C02003 V=800.0 PL=0
MOVL C02004 V=800.0 PL=0
MOVL C02005 V=800.0 PL=0
MOVL C02006 V=800.0 PL=0
MOVL C02007 V=800.0 PL=0
MOVL C02008 V=800.0 PL=0
MOVL C02009 V=800.0 PL=0
MOVL C02010 V=800.0 PL=0
MOVL C02011 V=800.0 PL=0
MOVL C02012 V=800.0 PL=0
MOVL C02013 V=800.0 PL=0
MOVL C02014 V=800.0 PL=0
MOVL C02015 V=800.0 PL=0
MOVL C02016 V=800.0 PL=0
MOVL C02017 V=800.0 PL=0
MOVL C02018 V=800.0 PL=0
MOVL C02019 V=800.0 PL=0
MOVL C02020 V=800.0 PL=0
MOVL C02021 V=800.0 PL=0
MOVL C02022 V=800.0 PL=0
MOVL C02023 V=800.0 PL=0
MOVL C02024 V=800.0 PL=0
MOVL C02025 V=800.0 PL=0
MOVL C02026 V=800.0 PL=0
MOVL C02027 V=800.0 PL=0
MOVL C02028 V=800.0 PL=0
MOVL C02029 V=800.0 PL=0
MOVL C02030 V=800.0 PL=0
MOVL C02031 V=800.0 PL=0
MOVL C02032 V=800.0 PL=0
MOVL C02033 V=800.0 PL=0
MOVL C02034 V=800.0 PL=0
MOVL C02035 V=800.0 PL=0
MOVL C02036 V=800.0 PL=0
MOVL C02037 V=800.0 PL=0
MOVL C02038 V=800.0 PL=0
MOVL C02039 V=800.0 PL=0
MOVL C02040 V=800.0 PL=0
MOVL C02041 V=800.0 PL=0
